KUKA KRL program: MyProgram_089().src

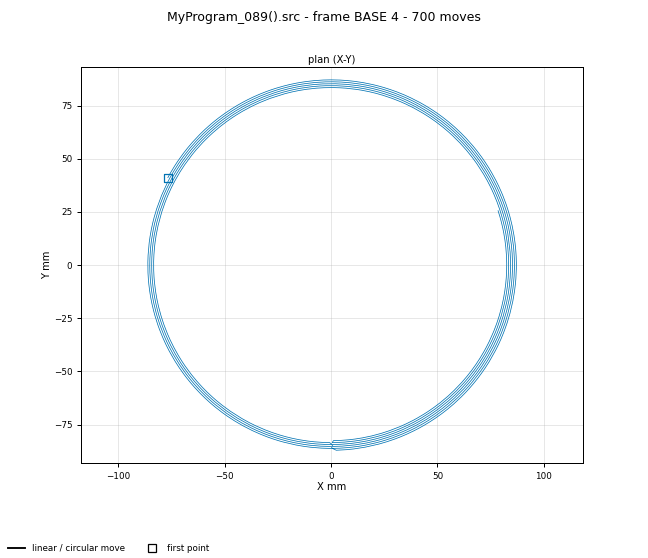
[picture p0: tool path of MyProgram_089().src in frame BASE 4, 700 of 700 moves have a stored position in this frame; points joined in program order, loops and branches not executed]
&ACCESS RVP
&REL 1
&PARAM TEMPLATE = C:\KRC\Roboter\Template\vorgabe
&PARAM EDITMASK = *
DEF MyProgram_089()
; ---- Setting reference (Base) ----
$BASE = BASE_DATA[4]

; --------------------------
; ---- Setting tool (TCP) ----
$TOOL = TOOL_DATA[3]
; --------------------------

$VEL.CP = VEL_APROX_PRINT
Startdeposition()
$VEL.CP = VEL_PRINT
LIN {X -76.7634,Y 41.1633,Z 86,A 146.3137,B 24.9093,C -2.1993,E1 24.8592,E2 298.6214} C_DIS
LIN {X -75.415,Y 43.5831,Z 86,A 144.1649,B 24.9096,C -2.1954,E1 24.8622,E2 300.7907} C_DIS
LIN {X -73.5045,Y 46.7342,Z 86,A 141.7026,B 24.9091,C -2.2011,E1 24.8658,E2 303.2518} C_DIS
LIN {X -72.1353,Y 48.8195,Z 86,A 139.243,B 24.9106,C -2.1828,E1 24.8698,E2 305.7674} C_DIS
LIN {X -69.4773,Y 52.5341,Z 86,A 137.1661,B 24.9078,C -2.2168,E1 24.8731,E2 307.7732} C_DIS
LIN {X -67.5267,Y 55.0186,Z 86,A 134.9351,B 24.9078,C -2.2179,E1 24.877,E2 310.012} C_DIS
LIN {X -65.1327,Y 57.8335,Z 86,A 132.6257,B 24.9069,C -2.2275,E1 24.8812,E2 312.3089} C_DIS
LIN {X -61.7541,Y 61.4278,Z 86,A 128.7956,B 24.9076,C -2.2188,E1 24.8887,E2 316.1763} C_DIS
LIN {X -59.3206,Y 63.7821,Z 86,A 127.0883,B 24.906,C -2.2388,E1 24.8921,E2 317.843} C_DIS
LIN {X -57.1612,Y 65.7228,Z 86,A 125.1507,B 24.9057,C -2.2423,E1 24.8962,E2 319.7798} C_DIS
LIN {X -54.8255,Y 67.6833,Z 86,A 123.2348,B 24.9051,C -2.2493,E1 24.9003,E2 321.6865} C_DIS
LIN {X -52.7347,Y 69.3257,Z 86,A 120.98,B 24.906,C -2.2384,E1 24.9054,E2 323.9752} C_DIS
LIN {X -49.8675,Y 71.4151,Z 86,A 118.3983,B 24.9062,C -2.236,E1 24.9113,E2 326.5717} C_DIS
LIN {X -46.7307,Y 73.5068,Z 86,A 116.0354,B 24.9055,C -2.244,E1 24.9168,E2 328.923} C_DIS
LIN {X -43.9125,Y 75.2237,Z 86,A 114.6023,B 24.9034,C -2.2693,E1 24.9202,E2 330.3002} C_DIS
LIN {X -41.4126,Y 76.6281,Z 86,A 112.4064,B 24.9039,C -2.2635,E1 24.9256,E2 332.5163} C_DIS
LIN {X -39.1074,Y 77.8311,Z 86,A 110.8125,B 24.9034,C -2.2696,E1 24.9295,E2 334.0999} C_DIS
LIN {X -36.432,Y 79.1182,Z 86,A 108.8082,B 24.9032,C -2.2711,E1 24.9346,E2 336.1056} C_DIS
LIN {X -33.5337,Y 80.3893,Z 86,A 106.7104,B 24.903,C -2.2736,E1 24.94,E2 338.2023} C_DIS
LIN {X -30.5403,Y 81.5736,Z 86,A 104.5603,B 24.9029,C -2.2755,E1 24.9456,E2 340.3526} C_DIS
LIN {X -28.173,Y 82.4213,Z 86,A 102.9203,B 24.9027,C -2.2779,E1 24.9499,E2 341.99} C_DIS
LIN {X -25.7542,Y 83.208,Z 86,A 101.1907,B 24.9027,C -2.2782,E1 24.9545,E2 343.722} C_DIS
LIN {X -22.1455,Y 84.2417,Z 86,A 98.7036,B 24.9025,C -2.2802,E1 24.9612,E2 346.2083} C_DIS
LIN {X -19.3941,Y 84.9162,Z 86,A 96.8617,B 24.9023,C -2.2825,E1 24.9662,E2 348.047} C_DIS
LIN {X -16.2854,Y 85.5668,Z 86,A 94.5826,B 24.9026,C -2.2785,E1 24.9725,E2 350.3382} C_DIS
LIN {X -12.7065,Y 86.172,Z 86,A 91.9605,B 24.9031,C -2.2731,E1 24.9797,E2 352.9755} C_DIS
LIN {X -8.1409,Y 86.7214,Z 86,A 89.5155,B 24.9014,C -2.2923,E1 24.9864,E2 355.3763} C_DIS
LIN {X -3.6843,Y 87.0246,Z 86,A 86.4266,B 24.9017,C -2.2888,E1 24.995,E2 358.4744} C_DIS
LIN {X 0.0247,Y 87.104,Z 86,A 83.8791,B 24.902,C -2.286,E1 25.0022,E2 361.0285} C_DIS
LIN {X 4.2369,Y 87.0001,Z 86,A 81.1959,B 24.9017,C -2.289,E1 25.0096,E2 363.7041} C_DIS
LIN {X 7.415,Y 86.7877,Z 86,A 78.9957,B 24.902,C -2.2856,E1 25.0158,E2 365.9111} C_DIS
LIN {X 11.0675,Y 86.3966,Z 86,A 76.481,B 24.9023,C -2.2822,E1 25.0228,E2 368.4322} C_DIS
LIN {X 15.0741,Y 85.789,Z 86,A 73.7549,B 24.9025,C -2.2794,E1 25.0303,E2 371.1621} C_DIS
LIN {X 19.4788,Y 84.8967,Z 86,A 71.0686,B 24.9019,C -2.2864,E1 25.0376,E2 373.8282} C_DIS
LIN {X 22.3755,Y 84.1802,Z 86,A 69.4228,B 24.9012,C -2.2953,E1 25.042,E2 375.4505} C_DIS
LIN {X 24.9228,Y 83.461,Z 86,A 67.479,B 24.9018,C -2.2876,E1 25.0472,E2 377.4091} C_DIS
LIN {X 27.8212,Y 82.5399,Z 86,A 65.4884,B 24.9019,C -2.2864,E1 25.0525,E2 379.399} C_DIS
LIN {X 30.9983,Y 81.4001,Z 86,A 63.1184,B 24.9025,C -2.2795,E1 25.0587,E2 381.7802} C_DIS
LIN {X 34.3976,Y 80.0241,Z 86,A 60.7222,B 24.9027,C -2.2775,E1 25.0649,E2 384.1756} C_DIS
LIN {X 37.4722,Y 78.6306,Z 86,A 58.5492,B 24.9027,C -2.2764,E1 25.0704,E2 386.3456} C_DIS
LIN {X 41.8101,Y 76.4125,Z 86,A 55.3258,B 24.9032,C -2.2716,E1 25.0784,E2 389.5714} C_DIS
LIN {X 45.0669,Y 74.5377,Z 86,A 53.0034,B 24.9031,C -2.2729,E1 25.0839,E2 391.8836} C_DIS
LIN {X 47.6981,Y 72.8823,Z 86,A 50.901,B 24.9035,C -2.2679,E1 25.0889,E2 393.9911} C_DIS
LIN {X 50.5181,Y 70.9562,Z 86,A 48.7009,B 24.9037,C -2.2657,E1 25.0939,E2 396.1888} C_DIS
LIN {X 52.437,Y 69.5502,Z 86,A 46.5187,B 24.9056,C -2.2427,E1 25.0989,E2 398.4176} C_DIS
LIN {X 55.2509,Y 67.3384,Z 86,A 44.6477,B 24.9047,C -2.2541,E1 25.1029,E2 400.2545} C_DIS
LIN {X 58.0486,Y 64.9401,Z 86,A 42.4392,B 24.9045,C -2.2566,E1 25.1075,E2 402.4484} C_DIS
LIN {X 61.0298,Y 62.1472,Z 86,A 39.1117,B 24.9067,C -2.2298,E1 25.1143,E2 405.8255} C_DIS
LIN {X 63.4116,Y 59.7146,Z 86,A 36.9778,B 24.9068,C -2.2284,E1 25.1184,E2 407.9534} C_DIS
LIN {X 66.661,Y 56.0663,Z 86,A 34.1325,B 24.9064,C -2.2333,E1 25.1235,E2 410.7742} C_DIS
LIN {X 68.5605,Y 53.7256,Z 86,A 32.4833,B 24.9059,C -2.2399,E1 25.1264,E2 412.4002} C_DIS
LIN {X 70.7515,Y 50.805,Z 86,A 30.1365,B 24.9062,C -2.2359,E1 25.1303,E2 414.7453} C_DIS
LIN {X 72.2333,Y 48.6749,Z 86,A 28.14,B 24.9074,C -2.2217,E1 25.1335,E2 416.7653} C_DIS
LIN {X 74.1305,Y 45.7351,Z 86,A 25.9158,B 24.9077,C -2.2184,E1 25.1368,E2 418.9861} C_DIS
LIN {X 75.4436,Y 43.5333,Z 86,A 24.1981,B 24.9081,C -2.2129,E1 25.1392,E2 420.7081} C_DIS
LIN {X 77.4348,Y 39.8846,Z 86,A 21.5317,B 24.9086,C -2.2077,E1 25.1427,E2 423.3726} C_DIS
LIN {X 78.666,Y 37.3985,Z 86,A 19.6238,B 24.9092,C -2.1998,E1 25.145,E2 425.289} C_DIS
LIN {X 80.0248,Y 34.3961,Z 86,A 17.5675,B 24.9094,C -2.1974,E1 25.1474,E2 427.3396} C_DIS
LIN {X 80.8251,Y 32.4701,Z 86,A 15.9985,B 24.9103,C -2.1867,E1 25.149,E2 428.9252} C_DIS
LIN {X 82.1991,Y 28.8126,Z 86,A 13.5608,B 24.9106,C -2.1838,E1 25.1513,E2 431.3563} C_DIS
LIN {X 83.2983,Y 25.4632,Z 86,A 11.4352,B 24.9106,C -2.1835,E1 25.1531,E2 433.4705} C_DIS
LIN {X 84.1421,Y 22.5169,Z 86,A 9.258,B 24.9115,C -2.1718,E1 25.1548,E2 435.6627} C_DIS
LIN {X 85.1237,Y 18.4612,Z 86,A 6.1814,B 24.9131,C -2.152,E1 25.1567,E2 438.7683} C_DIS
LIN {X 85.9827,Y 13.9294,Z 86,A 3.4164,B 24.9131,C -2.1518,E1 25.158,E2 441.5175} C_DIS
LIN {X 86.4939,Y 10.2803,Z 86,A 1.1857,B 24.9132,C -2.1509,E1 25.1588,E2 443.7373} C_DIS
LIN {X 86.8107,Y 7.1264,Z 86,A -0.8981,B 24.9138,C -2.1443,E1 25.1594,E2 445.8242} C_DIS
LIN {X 87.0169,Y 3.8645,Z 86,A -2.9324,B 24.914,C -2.1415,E1 25.1597,E2 447.853} C_DIS
LIN {X 87.0973,Y 1.0892,Z 86,A -5.0184,B 24.9152,C -2.1266,E1 25.1597,E2 449.9617} C_DIS
LIN {X 87.0851,Y -1.7482,Z 86,A -6.7904,B 24.9154,C -2.124,E1 25.1597,E2 451.7295} C_DIS
LIN {X 86.8701,Y -6.3796,Z 86,A -9.6702,B 24.9157,C -2.12,E1 25.1593,E2 454.6014} C_DIS
LIN {X 86.6351,Y -9.012,Z 86,A -11.4896,B 24.9164,C -2.1117,E1 25.1588,E2 456.4298} C_DIS
LIN {X 86.2143,Y -12.4087,Z 86,A -14.6166,B 24.9193,C -2.0744,E1 25.1575,E2 459.6264} C_DIS
LIN {X 85.4298,Y -16.9968,Z 86,A -16.5812,B 24.9171,C -2.1024,E1 25.1566,E2 461.5134} C_DIS
LIN {X 84.1155,Y -22.6153,Z 86,A -20.4328,B 24.9182,C -2.0884,E1 25.154,E2 465.3757} C_DIS
LIN {X 82.7404,Y -27.2225,Z 86,A -24.1318,B 24.9204,C -2.06,E1 25.1509,E2 469.1206} C_DIS
LIN {X 81.1349,Y -31.6862,Z 86,A -26.741,B 24.9198,C -2.0681,E1 25.1484,E2 471.6962} C_DIS
LIN {X 79.8438,Y -34.8112,Z 86,A -29.0086,B 24.9204,C -2.0598,E1 25.1459,E2 473.9709} C_DIS
LIN {X 78.7096,Y -37.3077,Z 86,A -30.8316,B 24.9209,C -2.0538,E1 25.1437,E2 475.7984} C_DIS
LIN {X 77.2971,Y -40.1528,Z 86,A -33.0905,B 24.9218,C -2.0418,E1 25.1409,E2 478.0737} C_DIS
LIN {X 74.3275,Y -45.4128,Z 86,A -36.9909,B 24.9225,C -2.0329,E1 25.1354,E2 481.975} C_DIS
LIN {X 72.2956,Y -48.5828,Z 86,A -39.2144,B 24.9224,C -2.0346,E1 25.132,E2 484.1832} C_DIS
LIN {X 70.6239,Y -50.9837,Z 86,A -41.1745,B 24.9229,C -2.0281,E1 25.1288,E2 486.1491} C_DIS
LIN {X 68.7131,Y -53.531,Z 86,A -43.1701,B 24.923,C -2.0259,E1 25.1254,E2 488.1404} C_DIS
LIN {X 66.9112,Y -55.7652,Z 86,A -45.1338,B 24.9236,C -2.0184,E1 25.1219,E2 490.1128} C_DIS
LIN {X 64.7202,Y -58.2943,Z 86,A -47.3545,B 24.9241,C -2.0121,E1 25.1178,E2 492.3384} C_DIS
LIN {X 62.938,Y -60.2143,Z 86,A -49.1674,B 24.9246,C -2.0048,E1 25.1143,E2 494.1607} C_DIS
LIN {X 61.1438,Y -62.0347,Z 86,A -51.6966,B 24.9271,C -1.9722,E1 25.1092,E2 496.7563} C_DIS
LIN {X 57.5449,Y -65.3877,Z 86,A -53.9194,B 24.9251,C -1.9987,E1 25.1047,E2 498.9075} C_DIS
LIN {X 55.0102,Y -67.5335,Z 86,A -55.8925,B 24.9249,C -2.001,E1 25.1005,E2 500.8676} C_DIS
LIN {X 53.3581,Y -68.8464,Z 86,A -57.4566,B 24.9256,C -1.9921,E1 25.097,E2 502.447} C_DIS
LIN {X 51.5911,Y -70.1801,Z 86,A -58.8812,B 24.9257,C -1.9901,E1 25.0938,E2 503.8712} C_DIS
LIN {X 48.9288,Y -72.0614,Z 86,A -60.9649,B 24.9259,C -1.9879,E1 25.089,E2 505.9531} C_DIS
LIN {X 46.5742,Y -73.6067,Z 86,A -62.9319,B 24.9265,C -1.9804,E1 25.0844,E2 507.9313} C_DIS
LIN {X 43.8648,Y -75.2527,Z 86,A -64.9876,B 24.9267,C -1.9776,E1 25.0795,E2 509.9874} C_DIS
LIN {X 41.2059,Y -76.7396,Z 86,A -66.9966,B 24.9269,C -1.974,E1 25.0745,E2 511.9992} C_DIS
LIN {X 38.8987,Y -77.9346,Z 86,A -69.3028,B 24.9286,C -1.9515,E1 25.0687,E2 514.3523} C_DIS
LIN {X 35.5869,Y -79.5014,Z 86,A -71.5732,B 24.9286,C -1.9524,E1 25.0629,E2 516.615} C_DIS
LIN {X 32.616,Y -80.7656,Z 86,A -73.1461,B 24.9274,C -1.9674,E1 25.0589,E2 518.1486} C_DIS
LIN {X 29.7282,Y -81.8725,Z 86,A -75.2929,B 24.9279,C -1.961,E1 25.0533,E2 520.306} C_DIS
LIN {X 26.2462,Y -83.0555,Z 86,A -77.5924,B 24.9279,C -1.962,E1 25.0472,E2 522.5989} C_DIS
LIN {X 22.4058,Y -84.1721,Z 86,A -80.4955,B 24.9287,C -1.9503,E1 25.0393,E2 525.5249} C_DIS
LIN {X 16.0344,Y -85.6151,Z 86,A -84.4685,B 24.9282,C -1.9569,E1 25.0286,E2 529.4771} C_DIS
LIN {X 10.7051,Y -86.4436,Z 86,A -88.1837,B 24.9288,C -1.949,E1 25.0182,E2 533.2075} C_DIS
LIN {X 7.4273,Y -86.7867,Z 86,A -90.3524,B 24.9288,C -1.9479,E1 25.0122,E2 535.3777} C_DIS
LIN {X 2.4408,Y -87.0687,Z 86,A -93.6388,B 24.929,C -1.9466,E1 25.003,E2 538.6661} C_DIS
LIN {X 2.4408,Y -87.0687,Z 86,A -93.6388,B 24.929,C -1.9466,E1 25.003,E2 538.6661} C_DIS
Enddeposition()
LIN {X 0.5553,Y -86.1888,Z 86,A -93.3756,B 24.9242,C -2.0102,E1 25.0042,E2 538.2522} C_DIS
Startdeposition()
$VEL.CP = VEL_PRINT
LIN {X 3.8721,Y -86.1086,Z 86,A -91.75,B 24.9256,C -1.9922,E1 25.0086,E2 536.6696} C_DIS
LIN {X 8.5981,Y -85.7663,Z 86,A -88.5017,B 24.9252,C -1.9969,E1 25.0177,E2 533.4119} C_DIS
LIN {X 13.0459,Y -85.2026,Z 86,A -85.1686,B 24.9242,C -2.0103,E1 25.027,E2 530.0497} C_DIS
LIN {X 16.2421,Y -84.6514,Z 86,A -82.1799,B 24.922,C -2.0396,E1 25.0354,E2 526.9952} C_DIS
LIN {X 21.4948,Y -83.4723,Z 86,A -80.2349,B 24.9258,C -1.9893,E1 25.0403,E2 525.1723} C_DIS
LIN {X 24.1077,Y -82.7557,Z 86,A -78.0283,B 24.9247,C -2.0045,E1 25.0463,E2 522.9333} C_DIS
LIN {X 26.2649,Y -82.0969,Z 86,A -76.4934,B 24.9244,C -2.0074,E1 25.0504,E2 521.3943} C_DIS
LIN {X 29.1197,Y -81.1289,Z 86,A -74.3708,B 24.924,C -2.0139,E1 25.056,E2 519.2606} C_DIS
LIN {X 33.6141,Y -79.3711,Z 86,A -71.1979,B 24.9237,C -2.0173,E1 25.0642,E2 516.087} C_DIS
LIN {X 37.2598,Y -77.7263,Z 86,A -68.3723,B 24.923,C -2.027,E1 25.0714,E2 513.2456} C_DIS
LIN {X 39.8478,Y -76.4326,Z 86,A -65.8675,B 24.9212,C -2.0498,E1 25.0778,E2 510.6938} C_DIS
LIN {X 43.6555,Y -74.323,Z 86,A -63.7162,B 24.9227,C -2.0299,E1 25.0828,E2 508.5961} C_DIS
LIN {X 46.5967,Y -72.5149,Z 86,A -61.6607,B 24.923,C -2.0262,E1 25.0876,E2 506.556} C_DIS
LIN {X 49.1239,Y -70.8273,Z 86,A -59.6458,B 24.9227,C -2.03,E1 25.0923,E2 504.5388} C_DIS
LIN {X 52.7293,Y -68.1858,Z 86,A -56.395,B 24.9215,C -2.0457,E1 25.0996,E2 501.2625} C_DIS
LIN {X 55.5568,Y -65.9038,Z 86,A -54.1006,B 24.9215,C -2.047,E1 25.1045,E2 498.9741} C_DIS
LIN {X 59.5946,Y -62.2747,Z 86,A -50.5714,B 24.921,C -2.0526,E1 25.1118,E2 495.4456} C_DIS
LIN {X 62.0674,Y -59.8105,Z 86,A -48.2048,B 24.9204,C -2.0599,E1 25.1164,E2 493.0721} C_DIS
LIN {X 64.5863,Y -57.0836,Z 86,A -45.8968,B 24.9204,C -2.0606,E1 25.1207,E2 490.7727} C_DIS
LIN {X 66.5451,Y -54.7865,Z 86,A -43.5845,B 24.9192,C -2.0764,E1 25.1249,E2 488.4338} C_DIS
LIN {X 70.0716,Y -50.1962,Z 86,A -40.0232,B 24.9192,C -2.0768,E1 25.1309,E2 484.8884} C_DIS
LIN {X 71.8513,Y -47.614,Z 86,A -37.3481,B 24.917,C -2.1031,E1 25.1351,E2 482.1645} C_DIS
LIN {X 73.7236,Y -44.6599,Z 86,A -35.9077,B 24.9189,C -2.079,E1 25.1371,E2 480.7883} C_DIS
LIN {X 76.3659,Y -39.9744,Z 86,A -32.2618,B 24.9179,C -2.0918,E1 25.1421,E2 477.1312} C_DIS
LIN {X 77.7306,Y -37.2508,Z 86,A -30.1507,B 24.9172,C -2.1008,E1 25.1447,E2 475.0102} C_DIS
LIN {X 79.2268,Y -33.9566,Z 86,A -27.6767,B 24.9165,C -2.1104,E1 25.1475,E2 472.527} C_DIS
LIN {X 80.2416,Y -31.4792,Z 86,A -25.4793,B 24.9149,C -2.1304,E1 25.1498,E2 470.2944} C_DIS
LIN {X 81.841,Y -27.055,Z 86,A -22.658,B 24.9149,C -2.1294,E1 25.1523,E2 467.4915} C_DIS
LIN {X 82.9666,Y -23.3714,Z 86,A -20.3616,B 24.9151,C -2.1282,E1 25.1541,E2 465.211} C_DIS
LIN {X 84.489,Y -17.0685,Z 86,A -16.1871,B 24.9143,C -2.137,E1 25.1568,E2 461.0398} C_DIS
LIN {X 85.4391,Y -11.3985,Z 86,A -12.4656,B 24.9137,C -2.1457,E1 25.1585,E2 457.3197} C_DIS
LIN {X 85.8101,Y -8.1449,Z 86,A -9.8442,B 24.9118,C -2.1681,E1 25.1593,E2 454.6609} C_DIS
LIN {X 86.0443,Y -5.1157,Z 86,A -7.3413,B 24.9099,C -2.1916,E1 25.1597,E2 452.1175} C_DIS
LIN {X 86.1848,Y -1.3715,Z 86,A -5.5151,B 24.9112,C -2.1762,E1 25.1597,E2 450.3384} C_DIS
LIN {X 86.1382,Y 3.1833,Z 86,A -2.2209,B 24.9096,C -2.1952,E1 25.1596,E2 447.0191} C_DIS
LIN {X 85.9696,Y 6.2509,Z 86,A -0.4717,B 24.9099,C -2.1914,E1 25.1592,E2 445.2891} C_DIS
LIN {X 85.6888,Y 9.3393,Z 86,A 1.541,B 24.9095,C -2.1962,E1 25.1587,E2 443.277} C_DIS
LIN {X 84.8873,Y 14.9631,Z 86,A 4.9917,B 24.9095,C -2.1967,E1 25.1573,E2 439.8454} C_DIS
LIN {X 83.9417,Y 19.5828,Z 86,A 7.9872,B 24.9091,C -2.2016,E1 25.1556,E2 436.8559} C_DIS
LIN {X 83.4156,Y 21.7157,Z 86,A 9.9382,B 24.9073,C -2.223,E1 25.1542,E2 434.8657} C_DIS
LIN {X 82.4756,Y 25.0536,Z 86,A 12.208,B 24.9068,C -2.2287,E1 25.1524,E2 432.5955} C_DIS
LIN {X 81.485,Y 28.1081,Z 86,A 14.3003,B 24.9064,C -2.2335,E1 25.1506,E2 430.5035} C_DIS
LIN {X 80.715,Y 30.2464,Z 86,A 16.6699,B 24.9035,C -2.2678,E1 25.1482,E2 428.0662} C_DIS
LIN {X 79.0291,Y 34.4103,Z 86,A 18.6301,B 24.9058,C -2.2408,E1 25.1461,E2 426.1805} C_DIS
LIN {X 77.8734,Y 36.9535,Z 86,A 21.6178,B 24.902,C -2.285,E1 25.1424,E2 423.1043} C_DIS
LIN {X 75.6326,Y 41.3454,Z 86,A 23.855,B 24.9044,C -2.258,E1 25.1395,E2 420.9428} C_DIS
LIN {X 74.0596,Y 44.1012,Z 86,A 26.2172,B 24.9031,C -2.2722,E1 25.1362,E2 418.559} C_DIS
LIN {X 72.0182,Y 47.3609,Z 86,A 28.3952,B 24.9037,C -2.2659,E1 25.1329,E2 416.4069} C_DIS
LIN {X 70.4033,Y 49.7312,Z 86,A 30.7155,B 24.9021,C -2.2848,E1 25.1291,E2 414.0535} C_DIS
LIN {X 67.5766,Y 53.5076,Z 86,A 33.5411,B 24.9023,C -2.2818,E1 25.1244,E2 411.2482} C_DIS
LIN {X 65.6319,Y 55.8759,Z 86,A 35.6341,B 24.9018,C -2.2884,E1 25.1206,E2 409.1492} C_DIS
LIN {X 61.1648,Y 60.7336,Z 86,A 39.729,B 24.9018,C -2.2882,E1 25.1128,E2 405.0727} C_DIS
LIN {X 59.7975,Y 62.0799,Z 86,A 41.3725,B 24.9005,C -2.3031,E1 25.1095,E2 403.4007} C_DIS
LIN {X 56.9904,Y 64.6676,Z 86,A 43.7106,B 24.9006,C -2.3015,E1 25.1046,E2 401.0759} C_DIS
LIN {X 54.6012,Y 66.6975,Z 86,A 46.2078,B 24.8991,C -2.3192,E1 25.0992,E2 398.5463} C_DIS
LIN {X 50.4399,Y 69.8976,Z 86,A 49.1243,B 24.9002,C -2.3063,E1 25.0928,E2 395.6709} C_DIS
LIN {X 47.8883,Y 71.6705,Z 86,A 51.2386,B 24.8998,C -2.3112,E1 25.0879,E2 393.552} C_DIS
LIN {X 45.1615,Y 73.4187,Z 86,A 53.8543,B 24.8982,C -2.3298,E1 25.0816,E2 390.9008} C_DIS
LIN {X 41.1371,Y 75.7456,Z 86,A 57.0566,B 24.8975,C -2.3377,E1 25.0738,E2 387.689} C_DIS
LIN {X 38.1933,Y 77.2719,Z 86,A 59.235,B 24.8973,C -2.3396,E1 25.0683,E2 385.512} C_DIS
LIN {X 35.2475,Y 78.6594,Z 86,A 60.7706,B 24.8989,C -2.3216,E1 25.0645,E2 384.0229} C_DIS
LIN {X 30.2889,Y 80.6989,Z 86,A 64.5187,B 24.898,C -2.3311,E1 25.0548,E2 380.2607} C_DIS
LIN {X 26.7118,Y 81.9523,Z 86,A 66.9481,B 24.8981,C -2.3303,E1 25.0484,E2 377.838} C_DIS
LIN {X 23.5489,Y 82.9163,Z 86,A 69.1096,B 24.8981,C -2.3307,E1 25.0426,E2 375.6792} C_DIS
LIN {X 20.0579,Y 83.8301,Z 86,A 71.5045,B 24.898,C -2.332,E1 25.0361,E2 373.2849} C_DIS
LIN {X 16.8841,Y 84.5269,Z 86,A 74.238,B 24.8963,C -2.3512,E1 25.0285,E2 370.5092} C_DIS
LIN {X 13.6155,Y 85.1145,Z 86,A 76.0994,B 24.8972,C -2.3409,E1 25.0234,E2 368.674} C_DIS
LIN {X 9.149,Y 85.7087,Z 86,A 78.519,B 24.8987,C -2.3235,E1 25.0169,E2 366.2978} C_DIS
LIN {X 4.6296,Y 86.0711,Z 86,A 81.8771,B 24.8978,C -2.3343,E1 25.0074,E2 362.9155} C_DIS
LIN {X 0.939,Y 86.1897,Z 86,A 84.7013,B 24.8968,C -2.3455,E1 24.9995,E2 360.0652} C_DIS
LIN {X -2.6768,Y 86.1539,Z 86,A 86.8743,B 24.8975,C -2.3377,E1 24.9935,E2 357.9106} C_DIS
LIN {X -7.7582,Y 85.8458,Z 86,A 89.7735,B 24.8989,C -2.3214,E1 24.9855,E2 355.0489} C_DIS
LIN {X -12.4441,Y 85.2931,Z 86,A 93.1212,B 24.8985,C -2.3259,E1 24.9762,E2 351.6881} C_DIS
LIN {X -14.9601,Y 84.8878,Z 86,A 94.9954,B 24.8981,C -2.3302,E1 24.971,E2 349.8021} C_DIS
LIN {X -18.1469,Y 84.2639,Z 86,A 97.1348,B 24.8983,C -2.3278,E1 24.9651,E2 347.6658} C_DIS
LIN {X -21.1295,Y 83.5662,Z 86,A 99.1946,B 24.8984,C -2.3266,E1 24.9596,E2 345.6061} C_DIS
LIN {X -24.0255,Y 82.781,Z 86,A 101.3524,B 24.8982,C -2.3294,E1 24.9537,E2 343.4382} C_DIS
LIN {X -26.6719,Y 81.9652,Z 86,A 103.5921,B 24.8973,C -2.3393,E1 24.9477,E2 341.1709} C_DIS
LIN {X -29.8506,Y 80.8623,Z 86,A 105.0252,B 24.8997,C -2.3124,E1 24.9441,E2 339.7989} C_DIS
LIN {X -33.387,Y 79.4668,Z 86,A 107.7798,B 24.8994,C -2.3157,E1 24.9369,E2 337.0305} C_DIS
LIN {X -36.226,Y 78.2136,Z 86,A 110.2294,B 24.8987,C -2.324,E1 24.9306,E2 334.5549} C_DIS
LIN {X -39.9,Y 76.4051,Z 86,A 112.6449,B 24.8998,C -2.3106,E1 24.9247,E2 332.1649} C_DIS
LIN {X -42.7024,Y 74.8748,Z 86,A 114.9169,B 24.8998,C -2.3113,E1 24.9191,E2 329.8846} C_DIS
LIN {X -46.4038,Y 72.6387,Z 86,A 117.9459,B 24.8998,C -2.3105,E1 24.9119,E2 326.848} C_DIS
LIN {X -50.3519,Y 69.9605,Z 86,A 121.2138,B 24.9001,C -2.307,E1 24.9045,E2 323.5773} C_DIS
LIN {X -53.9354,Y 67.2371,Z 86,A 124.0774,B 24.901,C -2.2969,E1 24.8982,E2 320.7271} C_DIS
LIN {X -57.9428,Y 63.8161,Z 86,A 127.9034,B 24.9009,C -2.2984,E1 24.8902,E2 316.8825} C_DIS
LIN {X -60.3048,Y 61.5865,Z 86,A 129.7077,B 24.9022,C -2.283,E1 24.8866,E2 315.1073} C_DIS
LIN {X -63.3063,Y 58.4954,Z 86,A 132.768,B 24.9023,C -2.2816,E1 24.8807,E2 312.0369} C_DIS
LIN {X -66.4209,Y 54.936,Z 86,A 135.8403,B 24.9032,C -2.2715,E1 24.8752,E2 308.9748} C_DIS
LIN {X -69.3278,Y 51.2196,Z 86,A 139.1812,B 24.9034,C -2.269,E1 24.8696,E2 305.6239} C_DIS
LIN {X -71.7307,Y 47.7969,Z 86,A 141.7923,B 24.9045,C -2.2565,E1 24.8655,E2 303.0296} C_DIS
LIN {X -74.0479,Y 44.1209,Z 86,A 144.4199,B 24.9058,C -2.2409,E1 24.8617,E2 300.4256} C_DIS
LIN {X -75.5519,Y 41.4942,Z 86,A 146.4376,B 24.9063,C -2.2353,E1 24.8589,E2 298.4108} C_DIS
LIN {X -77.1803,Y 38.3781,Z 86,A 149.1153,B 24.906,C -2.2381,E1 24.8555,E2 295.7122} C_DIS
LIN {X -79.6902,Y 32.8523,Z 86,A 152.9138,B 24.9076,C -2.2193,E1 24.8513,E2 291.9377} C_DIS
LIN {X -82.0216,Y 26.4975,Z 86,A 157.3186,B 24.909,C -2.2027,E1 24.8472,E2 287.5473} C_DIS
LIN {X -83.2516,Y 22.3349,Z 86,A 160.1807,B 24.9098,C -2.1931,E1 24.845,E2 284.6918} C_DIS
LIN {X -83.8659,Y 19.9107,Z 86,A 161.8913,B 24.9101,C -2.1892,E1 24.8438,E2 282.9804} C_DIS
LIN {X -84.5406,Y 16.8172,Z 86,A 164.0758,B 24.9105,C -2.1847,E1 24.8426,E2 280.7937} C_DIS
LIN {X -85.1512,Y 13.3779,Z 86,A 166.3693,B 24.9111,C -2.1766,E1 24.8415,E2 278.506} C_DIS
LIN {X -85.5596,Y 10.4597,Z 86,A 168.8152,B 24.9105,C -2.184,E1 24.8407,E2 276.0278} C_DIS
LIN {X -86.0761,Y 4.5397,Z 86,A 172.468,B 24.9122,C -2.163,E1 24.8399,E2 272.4032} C_DIS
LIN {X -86.1868,Y 1.2662,Z 86,A 174.9812,B 24.912,C -2.1655,E1 24.8398,E2 269.8688} C_DIS
LIN {X -86.1179,Y -3.6564,Z 86,A 177.7256,B 24.9141,C -2.1402,E1 24.84,E2 267.1683} C_DIS
LIN {X -85.9343,Y -6.7062,Z 86,A 179.531,B 24.9151,C -2.1275,E1 24.8403,E2 265.3824} C_DIS
LIN {X -85.7225,Y -9.0176,Z 86,A -178.321,B 24.9141,C -2.1396,E1 24.8409,E2 263.1927} C_DIS
LIN {X -85.3543,Y -12.0133,Z 86,A -176.5494,B 24.9152,C -2.1267,E1 24.8416,E2 261.4412} C_DIS
LIN {X -84.8694,Y -15.0628,Z 86,A -174.5012,B 24.9157,C -2.1202,E1 24.8425,E2 259.3964} C_DIS
LIN {X -84.2966,Y -17.997,Z 86,A -172.3818,B 24.9159,C -2.1178,E1 24.8437,E2 257.2703} C_DIS
LIN {X -83.5833,Y -21.0633,Z 86,A -170.3524,B 24.9165,C -2.1096,E1 24.845,E2 255.2486} C_DIS
LIN {X -82.8564,Y -23.7602,Z 86,A -168.5401,B 24.9171,C -2.1027,E1 24.8464,E2 253.4421} C_DIS
LIN {X -81.5811,Y -27.8257,Z 86,A -165.8313,B 24.918,C -2.0908,E1 24.8487,E2 250.7461} C_DIS
LIN {X -80.6988,Y -30.2891,Z 86,A -163.4949,B 24.9171,C -2.1027,E1 24.851,E2 248.3682} C_DIS
LIN {X -79.0848,Y -34.2824,Z 86,A -160.9313,B 24.9184,C -2.086,E1 24.8537,E2 245.8303} C_DIS
LIN {X -77.66,Y -37.3977,Z 86,A -158.709,B 24.919,C -2.078,E1 24.8564,E2 243.6149} C_DIS
LIN {X -76.0791,Y -40.5191,Z 86,A -156.2198,B 24.9192,C -2.0764,E1 24.8596,E2 241.1164} C_DIS
LIN {X -73.3035,Y -45.3475,Z 86,A -152.5489,B 24.92,C -2.0657,E1 24.8648,E2 237.452} C_DIS
LIN {X -71.4037,Y -48.2823,Z 86,A -149.5854,B 24.919,C -2.0784,E1 24.8695,E2 234.4433} C_DIS
LIN {X -69.1658,Y -51.4386,Z 86,A -147.9305,B 24.9215,C -2.0454,E1 24.8721,E2 232.8591} C_DIS
LIN {X -67.8726,Y -53.1331,Z 86,A -146.283,B 24.9213,C -2.0487,E1 24.8749,E2 231.1959} C_DIS
LIN {X -66.0712,Y -55.3569,Z 86,A -144.4081,B 24.9217,C -2.0435,E1 24.8782,E2 229.3247} C_DIS
LIN {X -64.149,Y -57.5724,Z 86,A -142.1609,B 24.9214,C -2.0478,E1 24.8824,E2 227.0571} C_DIS
LIN {X -61.8419,Y -60.0445,Z 86,A -140.0048,B 24.9219,C -2.0403,E1 24.8866,E2 224.9097} C_DIS
LIN {X -59.1443,Y -62.7026,Z 86,A -137.6562,B 24.9227,C -2.0302,E1 24.8913,E2 222.5755} C_DIS
LIN {X -56.9275,Y -64.7226,Z 86,A -135.6333,B 24.9229,C -2.0271,E1 24.8955,E2 220.5518} C_DIS
LIN {X -54.6919,Y -66.6235,Z 86,A -133.162,B 24.922,C -2.0389,E1 24.9009,E2 218.0429} C_DIS
LIN {X -51.3251,Y -69.2506,Z 86,A -130.7507,B 24.9234,C -2.0212,E1 24.9062,E2 215.6652} C_DIS
LIN {X -48.7319,Y -71.0992,Z 86,A -128.2162,B 24.9227,C -2.0303,E1 24.9121,E2 213.1004} C_DIS
LIN {X -45.396,Y -73.2732,Z 86,A -126.0301,B 24.9241,C -2.0124,E1 24.9171,E2 210.9499} C_DIS
LIN {X -41.5678,Y -75.5116,Z 86,A -122.8318,B 24.9238,C -2.0159,E1 24.925,E2 207.734} C_DIS
LIN {X -37.0249,Y -77.8392,Z 86,A -118.8609,B 24.9228,C -2.0295,E1 24.935,E2 203.7203} C_DIS
LIN {X -33.2317,Y -79.5323,Z 86,A -117.0231,B 24.9251,C -1.9982,E1 24.9396,E2 201.9526} C_DIS
LIN {X -30.004,Y -80.8063,Z 86,A -114.7164,B 24.9253,C -1.9961,E1 24.9456,E2 199.6462} C_DIS
LIN {X -27.1972,Y -81.793,Z 86,A -112.6645,B 24.9253,C -1.9967,E1 24.951,E2 197.5887} C_DIS
LIN {X -24.5686,Y -82.6199,Z 86,A -111.0332,B 24.9258,C -1.9892,E1 24.9553,E2 195.9724} C_DIS
LIN {X -22.4455,Y -83.2218,Z 86,A -109.3372,B 24.9253,C -1.9954,E1 24.9599,E2 194.2592} C_DIS
LIN {X -16.4006,Y -84.6209,Z 86,A -104.5942,B 24.924,C -2.0129,E1 24.973,E2 189.4687} C_DIS
LIN {X -13.011,Y -85.208,Z 86,A -102.9095,B 24.9255,C -1.9933,E1 24.9775,E2 187.8292} C_DIS
LIN {X -9.6911,Y -85.6496,Z 86,A -100.2271,B 24.9244,C -2.0073,E1 24.9851,E2 185.1115} C_DIS
LIN {X -4.4354,Y -86.0819,Z 86,A -97.1375,B 24.9254,C -1.9942,E1 24.9936,E2 182.0521} C_DIS
LIN {X -1.4013,Y -86.1843,Z 86,A -95.1006,B 24.9254,C -1.9951,E1 24.9993,E2 180.0127} C_DIS
LIN {X 0.5553,Y -86.1888,Z 86,A -93.3733,B 24.9243,C -2.0092,E1 25.0042,E2 178.2522} C_DIS
Enddeposition()
LIN {X 0.5553,Y -86.1888,Z 86,A -93.3733,B 24.9243,C -2.0092,E1 25.0042,E2 178.2522} C_DIS
Startdeposition()
$VEL.CP = VEL_PRINT
LIN {X 0.0638,Y -85.2896,Z 86,A -95.0303,B 24.9263,C -1.9827,E1 24.9994,E2 179.9719} C_DIS
LIN {X -4.8185,Y -85.1522,Z 86,A -98.2795,B 24.9263,C -1.9833,E1 24.9903,E2 183.2202} C_DIS
LIN {X -9.8423,Y -84.7186,Z 86,A -101.7537,B 24.9264,C -1.9808,E1 24.9807,E2 186.702} C_DIS
LIN {X -13.052,Y -84.2838,Z 86,A -104.4129,B 24.9275,C -1.9666,E1 24.9732,E2 189.3971} C_DIS
LIN {X -17.5571,Y -83.4627,Z 86,A -107.3505,B 24.9271,C -1.972,E1 24.9652,E2 192.3252} C_DIS
LIN {X -21.0062,Y -82.6614,Z 86,A -109.4522,B 24.9264,C -1.9816,E1 24.9595,E2 194.407} C_DIS
LIN {X -24.1919,Y -81.7855,Z 86,A -111.7583,B 24.9264,C -1.9805,E1 24.9533,E2 196.7195} C_DIS
LIN {X -27.8379,Y -80.6185,Z 86,A -114.0739,B 24.9257,C -1.9902,E1 24.9472,E2 199.0165} C_DIS
LIN {X -31.2159,Y -79.3705,Z 86,A -116.6127,B 24.9258,C -1.9888,E1 24.9406,E2 201.5637} C_DIS
LIN {X -35.0892,Y -77.7358,Z 86,A -119.331,B 24.9254,C -1.9949,E1 24.9336,E2 204.2738} C_DIS
LIN {X -37.3292,Y -76.6866,Z 86,A -121.5443,B 24.9264,C -1.9806,E1 24.9279,E2 206.5268} C_DIS
LIN {X -42.0382,Y -74.2092,Z 86,A -124.8702,B 24.9256,C -1.9926,E1 24.9198,E2 209.8336} C_DIS
LIN {X -45.1121,Y -72.3811,Z 86,A -128.1839,B 24.9272,C -1.97,E1 24.9118,E2 213.2116} C_DIS
LIN {X -49.0863,Y -69.7488,Z 86,A -130.1888,B 24.9243,C -2.0095,E1 24.9074,E2 215.129} C_DIS
LIN {X -54.5258,Y -65.5824,Z 86,A -134.5846,B 24.9232,C -2.0237,E1 24.8977,E2 219.5072} C_DIS
LIN {X -56.2412,Y -64.1176,Z 86,A -136.5962,B 24.9241,C -2.0123,E1 24.8934,E2 221.5537} C_DIS
LIN {X -58.8003,Y -61.781,Z 86,A -139.048,B 24.924,C -2.0135,E1 24.8884,E2 224.0127} C_DIS
LIN {X -61.7393,Y -58.8438,Z 86,A -142.4329,B 24.9248,C -2.0027,E1 24.8817,E2 227.4378} C_DIS
LIN {X -64.3364,Y -55.9907,Z 86,A -144.1581,B 24.9225,C -2.0329,E1 24.8787,E2 229.0989} C_DIS
LIN {X -66.1077,Y -53.8883,Z 86,A -146.1549,B 24.9225,C -2.0329,E1 24.8751,E2 231.1048} C_DIS
LIN {X -68.0446,Y -51.4208,Z 86,A -149.5164,B 24.9248,C -2.0033,E1 24.8693,E2 234.5532} C_DIS
LIN {X -71.2147,Y -46.9316,Z 86,A -151.4819,B 24.9204,C -2.0604,E1 24.8664,E2 236.3921} C_DIS
LIN {X -74.182,Y -42.0876,Z 86,A -156.0004,B 24.9211,C -2.0508,E1 24.8598,E2 240.9568} C_DIS
LIN {X -76.1143,Y -38.4819,Z 86,A -158.4984,B 24.92,C -2.0652,E1 24.8566,E2 243.4338} C_DIS
LIN {X -77.2573,Y -36.131,Z 86,A -160.2995,B 24.9197,C -2.0689,E1 24.8544,E2 245.2359} C_DIS
LIN {X -78.4356,Y -33.4982,Z 86,A -162.3186,B 24.9195,C -2.0721,E1 24.8521,E2 247.2584} C_DIS
LIN {X -80.3764,Y -28.5278,Z 86,A -166.7962,B 24.9206,C -2.0583,E1 24.8477,E2 251.7943} C_DIS
LIN {X -81.7222,Y -24.4051,Z 86,A -168.6787,B 24.9177,C -2.095,E1 24.8463,E2 253.6001} C_DIS
LIN {X -82.4208,Y -21.9324,Z 86,A -170.6054,B 24.9177,C -2.0947,E1 24.8448,E2 255.5386} C_DIS
LIN {X -83.3934,Y -17.8815,Z 86,A -173.5768,B 24.9174,C -2.0985,E1 24.843,E2 258.5182} C_DIS
LIN {X -84.0351,Y -14.5764,Z 86,A -175.6205,B 24.9164,C -2.1115,E1 24.8419,E2 260.5432} C_DIS
LIN {X -84.5081,Y -11.5208,Z 86,A -177.896,B 24.9164,C -2.1126,E1 24.841,E2 262.8296} C_DIS
LIN {X -84.9422,Y -7.6781,Z 86,A 179.6177,B 24.9154,C -2.1238,E1 24.8403,E2 265.304} C_DIS
LIN {X -85.2165,Y -3.5054,Z 86,A 176.9121,B 24.9145,C -2.1355,E1 24.8399,E2 267.9978} C_DIS
LIN {X -85.2858,Y -0.5852,Z 86,A 174.7845,B 24.9143,C -2.1373,E1 24.8398,E2 270.1341} C_DIS
LIN {X -85.2346,Y 3.0623,Z 86,A 172.1612,B 24.9141,C -2.1404,E1 24.84,E2 272.7657} C_DIS
LIN {X -84.9167,Y 7.9542,Z 86,A 168.7846,B 24.9134,C -2.1487,E1 24.8407,E2 276.1427} C_DIS
LIN {X -84.4928,Y 11.6279,Z 86,A 166.3777,B 24.9126,C -2.1587,E1 24.8415,E2 278.5401} C_DIS
LIN {X -83.6106,Y 16.837,Z 86,A 163.0035,B 24.9113,C -2.1748,E1 24.8432,E2 281.8961} C_DIS
LIN {X -82.9938,Y 19.6561,Z 86,A 160.9317,B 24.9111,C -2.1773,E1 24.8445,E2 283.9741} C_DIS
LIN {X -81.452,Y 25.2921,Z 86,A 157.5518,B 24.9089,C -2.2044,E1 24.847,E2 287.3088} C_DIS
LIN {X -80.2272,Y 28.9429,Z 86,A 154.1489,B 24.91,C -2.1901,E1 24.8501,E2 290.7652} C_DIS
LIN {X -78.709,Y 32.8493,Z 86,A 151.0605,B 24.91,C -2.1913,E1 24.8534,E2 293.868} C_DIS
LIN {X -77.4017,Y 35.8206,Z 86,A 149.3981,B 24.9082,C -2.2118,E1 24.8553,E2 295.4904} C_DIS
LIN {X -75.3176,Y 40.0183,Z 86,A 146.5097,B 24.9069,C -2.2282,E1 24.8589,E2 298.3553} C_DIS
LIN {X -74.2107,Y 42.0376,Z 86,A 144.7756,B 24.9069,C -2.2275,E1 24.8612,E2 300.1002} C_DIS
LIN {X -72.8212,Y 44.3981,Z 86,A 142.362,B 24.9078,C -2.2171,E1 24.8648,E2 302.551} C_DIS
LIN {X -70.331,Y 48.2486,Z 86,A 139.5577,B 24.9065,C -2.2331,E1 24.8691,E2 305.3311} C_DIS
LIN {X -67.6079,Y 51.9932,Z 86,A 136.0364,B 24.9067,C -2.2302,E1 24.875,E2 308.8762} C_DIS
LIN {X -65.5273,Y 54.5921,Z 86,A 134.3086,B 24.905,C -2.25,E1 24.878,E2 310.5649} C_DIS
LIN {X -62.64,Y 57.8815,Z 86,A 131.3108,B 24.9045,C -2.2558,E1 24.8836,E2 313.5623} C_DIS
LIN {X -60.0705,Y 60.5439,Z 86,A 128.5517,B 24.9047,C -2.2542,E1 24.8891,E2 316.3369} C_DIS
LIN {X -56.8442,Y 63.5834,Z 86,A 125.5741,B 24.9041,C -2.261,E1 24.8952,E2 319.3101} C_DIS
LIN {X -53.3562,Y 66.5389,Z 86,A 122.1504,B 24.9044,C -2.2579,E1 24.9026,E2 322.7543} C_DIS
LIN {X -50.4995,Y 68.7308,Z 86,A 120.7801,B 24.9014,C -2.2923,E1 24.9055,E2 324.0475} C_DIS
LIN {X -47.2058,Y 71.0338,Z 86,A 117.7163,B 24.9018,C -2.2873,E1 24.9126,E2 327.1336} C_DIS
LIN {X -45.0676,Y 72.4089,Z 86,A 115.4565,B 24.9029,C -2.2749,E1 24.9181,E2 329.43} C_DIS
LIN {X -41.2797,Y 74.6339,Z 86,A 113.0788,B 24.9011,C -2.2963,E1 24.9237,E2 331.7638} C_DIS
LIN {X -38.2433,Y 76.2347,Z 86,A 109.8713,B 24.9029,C -2.2745,E1 24.9319,E2 335.032} C_DIS
LIN {X -34.5131,Y 77.9947,Z 86,A 107.9225,B 24.9006,C -2.302,E1 24.9367,E2 336.92} C_DIS
LIN {X -31.7782,Y 79.1481,Z 86,A 105.4834,B 24.9014,C -2.292,E1 24.943,E2 339.3883} C_DIS
LIN {X -26.7179,Y 80.9969,Z 86,A 102.4491,B 24.8996,C -2.3134,E1 24.9509,E2 342.3776} C_DIS
LIN {X -23.2759,Y 82.0509,Z 86,A 99.9639,B 24.8996,C -2.3141,E1 24.9576,E2 344.8654} C_DIS
LIN {X -20.446,Y 82.8017,Z 86,A 97.8295,B 24.8998,C -2.3111,E1 24.9634,E2 347.0099} C_DIS
LIN {X -16.6371,Y 83.6514,Z 86,A 95.4207,B 24.899,C -2.3196,E1 24.9699,E2 349.4014} C_DIS
LIN {X -13.9481,Y 84.1402,Z 86,A 93.3706,B 24.8995,C -2.3147,E1 24.9756,E2 351.4654} C_DIS
LIN {X -8.6391,Y 84.8501,Z 86,A 89.9439,B 24.8988,C -2.3219,E1 24.985,E2 354.8774} C_DIS
LIN {X -3.8787,Y 85.2004,Z 86,A 86.74,B 24.8988,C -2.3233,E1 24.994,E2 358.0791} C_DIS
LIN {X 1.9869,Y 85.2663,Z 86,A 83.1066,B 24.8978,C -2.3334,E1 25.004,E2 361.6885} C_DIS
LIN {X 7.1389,Y 84.9898,Z 86,A 78.776,B 24.9001,C -2.3071,E1 25.0163,E2 366.0797} C_DIS
LIN {X 12.7239,Y 84.3345,Z 86,A 75.3756,B 24.8992,C -2.3178,E1 25.0256,E2 369.452} C_DIS
LIN {X 16.208,Y 83.7342,Z 86,A 72.9613,B 24.8994,C -2.3157,E1 25.0322,E2 371.8687} C_DIS
LIN {X 19.4304,Y 83.0459,Z 86,A 70.8698,B 24.8992,C -2.3183,E1 25.0379,E2 373.951} C_DIS
LIN {X 22.4504,Y 82.2808,Z 86,A 68.6711,B 24.8996,C -2.3138,E1 25.0439,E2 376.1571} C_DIS
LIN {X 25.7449,Y 81.3116,Z 86,A 66.0644,B 24.9005,C -2.3027,E1 25.0509,E2 378.7854} C_DIS
LIN {X 29.5632,Y 80.0016,Z 86,A 63.17,B 24.9012,C -2.2946,E1 25.0585,E2 381.693} C_DIS
LIN {X 32.6493,Y 78.7925,Z 86,A 61.5179,B 24.8999,C -2.3103,E1 25.0627,E2 383.3042} C_DIS
LIN {X 36.0115,Y 77.3129,Z 86,A 58.0902,B 24.9027,C -2.2774,E1 25.0716,E2 386.8009} C_DIS
LIN {X 40.1514,Y 75.2475,Z 86,A 56.1664,B 24.8998,C -2.3106,E1 25.0761,E2 388.6408} C_DIS
LIN {X 45.5927,Y 72.0808,Z 86,A 51.8844,B 24.9005,C -2.3028,E1 25.0864,E2 392.9283} C_DIS
LIN {X 47.6768,Y 70.7182,Z 86,A 50.0425,B 24.9012,C -2.2947,E1 25.0907,E2 394.7831} C_DIS
LIN {X 51.9947,Y 67.6067,Z 86,A 46.2167,B 24.9024,C -2.2805,E1 25.0994,E2 398.629} C_DIS
LIN {X 54.9204,Y 65.2543,Z 86,A 44.0026,B 24.902,C -2.2857,E1 25.1041,E2 400.8224} C_DIS
LIN {X 57.2369,Y 63.2318,Z 86,A 41.9142,B 24.9024,C -2.2809,E1 25.1085,E2 402.9138} C_DIS
LIN {X 59.4878,Y 61.1186,Z 86,A 39.5227,B 24.9036,C -2.2663,E1 25.1133,E2 405.3299} C_DIS
LIN {X 63.1728,Y 57.3012,Z 86,A 36.0011,B 24.9042,C -2.2599,E1 25.1201,E2 408.8513} C_DIS
LIN {X 65.6577,Y 54.4352,Z 86,A 33.8185,B 24.9037,C -2.266,E1 25.124,E2 411.0095} C_DIS
LIN {X 68.7165,Y 50.5191,Z 86,A 30.4814,B 24.9044,C -2.258,E1 25.1296,E2 414.3497} C_DIS
LIN {X 70.3346,Y 48.2434,Z 86,A 28.4728,B 24.9051,C -2.2489,E1 25.1329,E2 416.37} C_DIS
LIN {X 73.1557,Y 43.8478,Z 86,A 25.0088,B 24.9058,C -2.2412,E1 25.138,E2 419.8345} C_DIS
LIN {X 74.8969,Y 40.7993,Z 86,A 21.8581,B 24.9085,C -2.2088,E1 25.1423,E2 423.0454} C_DIS
LIN {X 76.911,Y 36.8618,Z 86,A 19.9188,B 24.9063,C -2.2347,E1 25.1446,E2 424.9131} C_DIS
LIN {X 77.9139,Y 34.6941,Z 86,A 17.1179,B 24.91,C -2.1904,E1 25.1479,E2 427.8032} C_DIS
LIN {X 79.8216,Y 30.0441,Z 86,A 15.2459,B 24.9067,C -2.2307,E1 25.1497,E2 429.5697} C_DIS
LIN {X 80.6729,Y 27.6804,Z 86,A 13.3746,B 24.9076,C -2.2196,E1 25.1514,E2 431.4569} C_DIS
LIN {X 81.4724,Y 25.2261,Z 86,A 11.4967,B 24.9084,C -2.2096,E1 25.153,E2 433.3477} C_DIS
LIN {X 82.3703,Y 22.1193,Z 86,A 9.3043,B 24.909,C -2.2023,E1 25.1547,E2 435.5447} C_DIS
LIN {X 83.1653,Y 18.9139,Z 86,A 6.3328,B 24.9117,C -2.1703,E1 25.1566,E2 438.5745} C_DIS
LIN {X 83.954,Y 15.0281,Z 86,A 3.9567,B 24.9115,C -2.1716,E1 25.1578,E2 440.9336} C_DIS
LIN {X 84.7481,Y 9.5902,Z 86,A 0.6912,B 24.9113,C -2.1744,E1 25.159,E2 444.1733} C_DIS
LIN {X 85.1136,Y 5.455,Z 86,A -2.0458,B 24.9119,C -2.1673,E1 25.1595,E2 446.9107} C_DIS
LIN {X 85.2677,Y 1.844,Z 86,A -4.6984,B 24.9131,C -2.152,E1 25.1598,E2 449.5838} C_DIS
LIN {X 85.2482,Y -2.6188,Z 86,A -7.9019,B 24.9145,C -2.1355,E1 25.1596,E2 452.8071} C_DIS
LIN {X 85.088,Y -5.8441,Z 86,A -10.2184,B 24.9154,C -2.1236,E1 25.1591,E2 455.138} C_DIS
LIN {X 84.7467,Y -9.6023,Z 86,A -11.9624,B 24.9139,C -2.1422,E1 25.1586,E2 456.8279} C_DIS
LIN {X 84.3881,Y -12.3649,Z 86,A -14.4449,B 24.9161,C -2.1155,E1 25.1576,E2 459.3586} C_DIS
LIN {X 83.847,Y -15.6216,Z 86,A -16.1807,B 24.9153,C -2.1247,E1 25.1568,E2 461.0625} C_DIS
LIN {X 82.5727,Y -21.3511,Z 86,A -20.2528,B 24.9167,C -2.1079,E1 25.1542,E2 465.1507} C_DIS
LIN {X 81.0374,Y -26.5927,Z 86,A -23.4345,B 24.9163,C -2.113,E1 25.1516,E2 468.3023} C_DIS
LIN {X 79.3896,Y -31.1674,Z 86,A -26.8754,B 24.9175,C -2.097,E1 25.1483,E2 471.7617} C_DIS
LIN {X 78.1915,Y -34.0616,Z 86,A -28.9985,B 24.9181,C -2.09,E1 25.146,E2 473.8897} C_DIS
LIN {X 76.2498,Y -38.2128,Z 86,A -32.1465,B 24.919,C -2.0784,E1 25.1422,E2 477.048} C_DIS
LIN {X 73.6123,Y -43.0753,Z 86,A -35.5256,B 24.919,C -2.079,E1 25.1377,E2 480.4081} C_DIS
LIN {X 70.8242,Y -47.5203,Z 86,A -39.0058,B 24.9196,C -2.0706,E1 25.1325,E2 483.8908} C_DIS
LIN {X 68.8318,Y -50.3617,Z 86,A -41.8424,B 24.9214,C -2.0472,E1 25.1278,E2 486.7687} C_DIS
LIN {X 66.4088,Y -53.5161,Z 86,A -44.2933,B 24.9214,C -2.0475,E1 25.1236,E2 489.2074} C_DIS
LIN {X 64.4495,Y -55.8612,Z 86,A -46.2916,B 24.9217,C -2.0441,E1 25.12,E2 491.2048} C_DIS
LIN {X 62.345,Y -58.2006,Z 86,A -48.8553,B 24.9232,C -2.0238,E1 25.115,E2 493.805} C_DIS
LIN {X 58.0117,Y -62.52,Z 86,A -52.688,B 24.9232,C -2.0232,E1 25.1074,E2 497.6232} C_DIS
LIN {X 54.7899,Y -65.3629,Z 86,A -55.948,B 24.9247,C -2.0044,E1 25.1004,E2 500.9149} C_DIS
LIN {X 52.1005,Y -67.5252,Z 86,A -57.8822,B 24.9241,C -2.0121,E1 25.0962,E2 502.8239} C_DIS
LIN {X 48.1237,Y -70.4156,Z 86,A -60.6867,B 24.9234,C -2.0217,E1 25.0899,E2 505.5959} C_DIS
LIN {X 44.781,Y -72.5869,Z 86,A -63.7024,B 24.9246,C -2.0055,E1 25.0827,E2 508.6401} C_DIS
LIN {X 40.1469,Y -75.2499,Z 86,A -66.985,B 24.9243,C -2.0091,E1 25.0748,E2 511.9044} C_DIS
LIN {X 35.5816,Y -77.513,Z 86,A -70.4372,B 24.9248,C -2.0027,E1 25.0661,E2 515.3627} C_DIS
LIN {X 30.8908,Y -79.4982,Z 86,A -73.7204,B 24.9248,C -2.0022,E1 25.0577,E2 518.6393} C_DIS
LIN {X 27.2451,Y -80.8196,Z 86,A -76.6853,B 24.926,C -1.9873,E1 25.0498,E2 521.6336} C_DIS
LIN {X 22.8394,Y -82.1743,Z 86,A -79.5274,B 24.9256,C -1.9919,E1 25.0422,E2 524.4598} C_DIS
LIN {X 20.9081,Y -82.6866,Z 86,A -81.9581,B 24.9283,C -1.9562,E1 25.0354,E2 526.9715} C_DIS
LIN {X 16.4992,Y -83.6781,Z 86,A -84.0692,B 24.9263,C -1.9825,E1 25.0298,E2 529.0174} C_DIS
LIN {X 11.3022,Y -84.5369,Z 86,A -87.6459,B 24.9266,C -1.9788,E1 25.0199,E2 532.5996} C_DIS
LIN {X 5.0835,Y -85.1376,Z 86,A -91.9232,B 24.9269,C -1.9742,E1 25.008,E2 536.8856} C_DIS
LIN {X 0.5378,Y -85.2804,Z 86,A -93.6627,B 24.9239,C -2.0145,E1 25.0035,E2 538.5288} C_DIS
Enddeposition()
LIN {X 0.5378,Y -85.2804,Z 86,A -93.6627,B 24.9239,C -2.0145,E1 25.0035,E2 538.5288} C_DIS
Startdeposition()
$VEL.CP = VEL_PRINT
LIN {X 0.8604,Y -84.3776,Z 86,A -93.0048,B 24.9217,C -2.0438,E1 25.0055,E2 537.8015} C_DIS
LIN {X 4.5186,Y -84.2603,Z 86,A -91.3231,B 24.9235,C -2.0195,E1 25.01,E2 536.1782} C_DIS
LIN {X 9.3897,Y -83.8583,Z 86,A -87.834,B 24.923,C -2.0265,E1 25.0197,E2 532.6744} C_DIS
LIN {X 12.5346,Y -83.4459,Z 86,A -85.6482,B 24.9228,C -2.029,E1 25.0258,E2 530.4847} C_DIS
LIN {X 16.7361,Y -82.7053,Z 86,A -82.1796,B 24.9212,C -2.0497,E1 25.0354,E2 526.971} C_DIS
LIN {X 20.2957,Y -81.9047,Z 86,A -80.4765,B 24.9229,C -2.0272,E1 25.0399,E2 525.3236} C_DIS
LIN {X 23.0574,Y -81.17,Z 86,A -77.9686,B 24.9214,C -2.0476,E1 25.0467,E2 522.7716} C_DIS
LIN {X 26.9343,Y -79.9672,Z 86,A -75.6677,B 24.9223,C -2.0362,E1 25.0528,E2 520.5021} C_DIS
LIN {X 30.6403,Y -78.6221,Z 86,A -72.4018,B 24.9205,C -2.0589,E1 25.0614,E2 517.1893} C_DIS
LIN {X 33.8524,Y -77.2932,Z 86,A -70.6119,B 24.9217,C -2.0438,E1 25.0659,E2 515.4396} C_DIS
LIN {X 39.1461,Y -74.7517,Z 86,A -66.7679,B 24.9215,C -2.0455,E1 25.0755,E2 511.6018} C_DIS
LIN {X 42.701,Y -72.7798,Z 86,A -62.9616,B 24.9185,C -2.0851,E1 25.0849,E2 507.7134} C_DIS
LIN {X 46.6345,Y -70.3241,Z 86,A -60.7454,B 24.9204,C -2.0601,E1 25.0899,E2 505.5634} C_DIS
LIN {X 50.3717,Y -67.6973,Z 86,A -57.7593,B 24.9202,C -2.0627,E1 25.0967,E2 502.5818} C_DIS
LIN {X 55.1412,Y -63.874,Z 86,A -53.5025,B 24.9192,C -2.0753,E1 25.1059,E2 498.3114} C_DIS
LIN {X 58.1265,Y -61.1679,Z 86,A -50.7355,B 24.9187,C -2.0827,E1 25.1116,E2 495.538} C_DIS
LIN {X 60.9841,Y -58.3202,Z 86,A -47.8642,B 24.9178,C -2.0938,E1 25.1172,E2 492.6527} C_DIS
LIN {X 63.7782,Y -55.2508,Z 86,A -44.3625,B 24.9154,C -2.1242,E1 25.1238,E2 489.0952} C_DIS
LIN {X 66.7024,Y -51.6822,Z 86,A -42.5614,B 24.9183,C -2.0874,E1 25.1268,E2 487.3893} C_DIS
LIN {X 69.6119,Y -47.6928,Z 86,A -38.8156,B 24.9165,C -2.1097,E1 25.1329,E2 483.609} C_DIS
LIN {X 71.0585,Y -45.5072,Z 86,A -36.8516,B 24.9156,C -2.121,E1 25.1359,E2 481.6283} C_DIS
LIN {X 73.0449,Y -42.2458,Z 86,A -34.055,B 24.9145,C -2.1353,E1 25.1399,E2 478.8122} C_DIS
LIN {X 75.1698,Y -38.3368,Z 86,A -31.7199,B 24.9156,C -2.1209,E1 25.1428,E2 476.5236} C_DIS
LIN {X 76.6326,Y -35.3235,Z 86,A -29.1369,B 24.9143,C -2.1381,E1 25.146,E2 473.9138} C_DIS
LIN {X 78.1103,Y -31.9218,Z 86,A -26.9516,B 24.9146,C -2.1344,E1 25.1483,E2 471.7491} C_DIS
LIN {X 79.5947,Y -28.016,Z 86,A -23.9319,B 24.9134,C -2.1493,E1 25.1513,E2 468.7111} C_DIS
LIN {X 80.9568,Y -23.796,Z 86,A -20.4569,B 24.9113,C -2.1746,E1 25.1542,E2 465.1962} C_DIS
LIN {X 82.574,Y -17.3753,Z 86,A -16.1883,B 24.9108,C -2.181,E1 25.1569,E2 460.9373} C_DIS
LIN {X 83.3666,Y -13.0474,Z 86,A -13.561,B 24.911,C -2.1782,E1 25.1581,E2 458.332} C_DIS
LIN {X 83.783,Y -10.033,Z 86,A -11.5878,B 24.9107,C -2.1816,E1 25.1588,E2 456.3624} C_DIS
LIN {X 84.178,Y -5.8556,Z 86,A -7.7796,B 24.9072,C -2.2236,E1 25.1596,E2 452.4776} C_DIS
LIN {X 84.3672,Y -1.5447,Z 86,A -5.7407,B 24.909,C -2.2024,E1 25.1598,E2 450.5009} C_DIS
LIN {X 84.351,Y 2.2802,Z 86,A -3.0946,B 24.9082,C -2.2123,E1 25.1597,E2 447.847} C_DIS
LIN {X 84.1535,Y 6.1899,Z 86,A -0.1139,B 24.9066,C -2.2318,E1 25.1591,E2 444.8381} C_DIS
LIN {X 83.0906,Y 14.704,Z 86,A 5.8411,B 24.9047,C -2.2544,E1 25.1568,E2 438.8649} C_DIS
LIN {X 82.439,Y 18.0004,Z 86,A 7.4625,B 24.906,C -2.2389,E1 25.1558,E2 437.2894} C_DIS
LIN {X 81.7601,Y 20.8691,Z 86,A 9.4972,B 24.9054,C -2.2462,E1 25.1545,E2 435.2494} C_DIS
LIN {X 80.8939,Y 24.008,Z 86,A 11.7545,B 24.9047,C -2.2544,E1 25.1527,E2 432.9857} C_DIS
LIN {X 79.9343,Y 27.0318,Z 86,A 14.1922,B 24.9033,C -2.2704,E1 25.1506,E2 430.524} C_DIS
LIN {X 78.93,Y 29.8372,Z 86,A 16.4028,B 24.9022,C -2.2826,E1 25.1484,E2 428.2967} C_DIS
LIN {X 77.7225,Y 32.8546,Z 86,A 18.1483,B 24.903,C -2.2733,E1 25.1465,E2 426.5827} C_DIS
LIN {X 76.2304,Y 36.1841,Z 86,A 21.483,B 24.8999,C -2.3093,E1 25.1425,E2 423.1811} C_DIS
LIN {X 74.1612,Y 40.2532,Z 86,A 23.6415,B 24.902,C -2.2859,E1 25.1397,E2 421.0891} C_DIS
LIN {X 72.3776,Y 43.3815,Z 86,A 27.0102,B 24.8987,C -2.3234,E1 25.1348,E2 417.6491} C_DIS
LIN {X 69.9114,Y 47.2505,Z 86,A 29.1002,B 24.901,C -2.297,E1 25.1317,E2 415.632} C_DIS
LIN {X 68.5746,Y 49.1708,Z 86,A 31.7719,B 24.8975,C -2.3371,E1 25.1272,E2 412.8783} C_DIS
LIN {X 65.6029,Y 53.0704,Z 86,A 34.027,B 24.9,C -2.3092,E1 25.1234,E2 410.6999} C_DIS
LIN {X 64.2123,Y 54.7447,Z 86,A 36.0561,B 24.8981,C -2.3308,E1 25.1197,E2 408.6288} C_DIS
LIN {X 61.9918,Y 57.2476,Z 86,A 37.5519,B 24.8999,C -2.3102,E1 25.1169,E2 407.1883} C_DIS
LIN {X 59.0267,Y 60.3009,Z 86,A 40.703,B 24.8986,C -2.3249,E1 25.1107,E2 404.0159} C_DIS
LIN {X 56.3447,Y 62.8131,Z 86,A 43.0689,B 24.8986,C -2.3257,E1 25.1059,E2 401.6577} C_DIS
LIN {X 54.061,Y 64.7892,Z 86,A 44.9877,B 24.8986,C -2.3254,E1 25.1018,E2 399.7472} C_DIS
LIN {X 51.7729,Y 66.6325,Z 86,A 47.4481,B 24.8969,C -2.3441,E1 25.0963,E2 397.2517} C_DIS
LIN {X 47.5462,Y 69.7112,Z 86,A 50.7063,B 24.8972,C -2.3406,E1 25.089,E2 394.0131} C_DIS
LIN {X 43.7237,Y 72.1697,Z 86,A 54.2757,B 24.8954,C -2.3609,E1 25.0804,E2 390.407} C_DIS
LIN {X 39.4024,Y 74.6168,Z 86,A 58.3436,B 24.893,C -2.3878,E1 25.0703,E2 386.2867} C_DIS
LIN {X 34.5347,Y 76.9908,Z 86,A 60.7912,B 24.8961,C -2.3526,E1 25.0643,E2 383.9288} C_DIS
LIN {X 32.2555,Y 77.9744,Z 86,A 62.5511,B 24.8958,C -2.3567,E1 25.0597,E2 382.1632} C_DIS
LIN {X 28.5839,Y 79.3932,Z 86,A 64.8831,B 24.8965,C -2.3486,E1 25.0537,E2 379.8556} C_DIS
LIN {X 25.2526,Y 80.5145,Z 86,A 67.5546,B 24.8955,C -2.3594,E1 25.0466,E2 377.1635} C_DIS
LIN {X 22.0684,Y 81.4444,Z 86,A 69.7899,B 24.8955,C -2.3604,E1 25.0406,E2 374.9296} C_DIS
LIN {X 18.9689,Y 82.2216,Z 86,A 71.8724,B 24.8955,C -2.3589,E1 25.0349,E2 372.8537} C_DIS
LIN {X 15.9614,Y 82.8579,Z 86,A 73.8176,B 24.8959,C -2.3554,E1 25.0296,E2 370.919} C_DIS
LIN {X 12.3541,Y 83.4735,Z 86,A 77.5207,B 24.8925,C -2.3939,E1 25.0192,E2 367.1282} C_DIS
LIN {X 7.6918,Y 84.03,Z 86,A 79.7477,B 24.8951,C -2.3646,E1 25.0132,E2 364.9722} C_DIS
LIN {X 2.5138,Y 84.3439,Z 86,A 83.0798,B 24.8956,C -2.3587,E1 25.0039,E2 361.6553} C_DIS
LIN {X -2.5268,Y 84.3435,Z 86,A 86.6124,B 24.8954,C -2.3612,E1 24.9941,E2 358.1166} C_DIS
LIN {X -5.1952,Y 84.2226,Z 86,A 88.6113,B 24.895,C -2.3661,E1 24.9884,E2 356.1055} C_DIS
LIN {X -9.0801,Y 83.8919,Z 86,A 91.5715,B 24.8942,C -2.3741,E1 24.9802,E2 353.1245} C_DIS
LIN {X -13.8261,Y 83.2409,Z 86,A 94.1693,B 24.8962,C -2.3524,E1 24.9731,E2 350.5761} C_DIS
LIN {X -16.73,Y 82.7065,Z 86,A 96.0409,B 24.8966,C -2.3469,E1 24.968,E2 348.7156} C_DIS
LIN {X -19.1989,Y 82.1684,Z 86,A 98.1571,B 24.8957,C -2.3572,E1 24.9622,E2 346.5723} C_DIS
LIN {X -22.526,Y 81.3205,Z 86,A 101.2619,B 24.8939,C -2.3777,E1 24.9537,E2 343.4139} C_DIS
LIN {X -26.504,Y 80.1123,Z 86,A 103.8784,B 24.8948,C -2.3682,E1 24.9468,E2 340.8152} C_DIS
LIN {X -29.7333,Y 78.9694,Z 86,A 106.0123,B 24.8955,C -2.3596,E1 24.9412,E2 338.6975} C_DIS
LIN {X -33.5048,Y 77.4447,Z 86,A 108.7332,B 24.896,C -2.3544,E1 24.9343,E2 335.9826} C_DIS
LIN {X -37.8113,Y 75.4364,Z 86,A 112.019,B 24.8963,C -2.351,E1 24.926,E2 332.6962} C_DIS
LIN {X -41.6311,Y 73.3981,Z 86,A 114.3651,B 24.8982,C -2.3289,E1 24.9204,E2 330.396} C_DIS
LIN {X -45.75,Y 70.9026,Z 86,A 118.7426,B 24.896,C -2.3546,E1 24.9099,E2 325.9434} C_DIS
LIN {X -49.4097,Y 68.4041,Z 86,A 120.841,B 24.8988,C -2.3225,E1 24.9052,E2 323.9143} C_DIS
LIN {X -52.777,Y 65.8407,Z 86,A 124.4275,B 24.8976,C -2.3367,E1 24.8973,E2 320.2809} C_DIS
LIN {X -55.5525,Y 63.5148,Z 86,A 126.2818,B 24.8995,C -2.3141,E1 24.8934,E2 318.4733} C_DIS
LIN {X -58.0419,Y 61.249,Z 86,A 128.2237,B 24.9008,C -2.2992,E1 24.8895,E2 316.5589} C_DIS
LIN {X -60.8682,Y 58.4405,Z 86,A 131.8541,B 24.8991,C -2.3186,E1 24.8823,E2 312.8668} C_DIS
LIN {X -63.2603,Y 55.8439,Z 86,A 133.6857,B 24.901,C -2.2967,E1 24.879,E2 311.0792} C_DIS
LIN {X -65.4655,Y 53.24,Z 86,A 137.3535,B 24.8983,C -2.3286,E1 24.8724,E2 307.318} C_DIS
LIN {X -69.0232,Y 48.5409,Z 86,A 140.0633,B 24.9023,C -2.2815,E1 24.8681,E2 304.7076} C_DIS
LIN {X -70.5221,Y 46.3342,Z 86,A 142.5959,B 24.901,C -2.2966,E1 24.8642,E2 302.1263} C_DIS
LIN {X -72.6129,Y 42.9834,Z 86,A 144.4873,B 24.9036,C -2.267,E1 24.8615,E2 300.2957} C_DIS
LIN {X -74.3873,Y 39.8364,Z 86,A 147.8178,B 24.9021,C -2.2842,E1 24.857,E2 296.9067} C_DIS
LIN {X -76.2413,Y 36.1614,Z 86,A 149.9125,B 24.9045,C -2.2565,E1 24.8545,E2 294.8666} C_DIS
LIN {X -78.0515,Y 32.0662,Z 86,A 152.9332,B 24.9053,C -2.2468,E1 24.8512,E2 291.8524} C_DIS
LIN {X -80.46,Y 25.4283,Z 86,A 157.6498,B 24.9067,C -2.2299,E1 24.8469,E2 287.1494} C_DIS
LIN {X -81.9923,Y 19.9367,Z 86,A 161.6562,B 24.9074,C -2.2214,E1 24.844,E2 283.1399} C_DIS
LIN {X -83.238,Y 13.8433,Z 86,A 166.1988,B 24.9078,C -2.2167,E1 24.8416,E2 278.5816} C_DIS
LIN {X -83.7698,Y 10.1458,Z 86,A 168.4888,B 24.9091,C -2.2019,E1 24.8407,E2 276.3134} C_DIS
LIN {X -84.1394,Y 6.3939,Z 86,A 170.7565,B 24.9104,C -2.1857,E1 24.8402,E2 274.0706} C_DIS
LIN {X -84.3114,Y 3.4379,Z 86,A 172.9699,B 24.9104,C -2.1848,E1 24.8399,E2 271.8461} C_DIS
LIN {X -84.3797,Y 0.3739,Z 86,A 175.6694,B 24.9096,C -2.1952,E1 24.8399,E2 269.1056} C_DIS
LIN {X -84.3283,Y -3.0144,Z 86,A 177.6556,B 24.9109,C -2.1792,E1 24.8399,E2 267.1458} C_DIS
LIN {X -84.1222,Y -6.6084,Z 86,A 179.8268,B 24.9122,C -2.1639,E1 24.8404,E2 264.9977} C_DIS
LIN {X -83.7382,Y -10.4022,Z 86,A -177.4155,B 24.9125,C -2.1604,E1 24.8412,E2 262.232} C_DIS
LIN {X -83.2013,Y -14.0628,Z 86,A -175.1614,B 24.9137,C -2.1455,E1 24.8422,E2 260.0001} C_DIS
LIN {X -82.4902,Y -17.7659,Z 86,A -171.7818,B 24.9125,C -2.1602,E1 24.8441,E2 256.5655} C_DIS
LIN {X -81.6897,Y -21.1426,Z 86,A -170.0007,B 24.9143,C -2.1371,E1 24.8453,E2 254.8291} C_DIS
LIN {X -80.9922,Y -23.6766,Z 86,A -167.807,B 24.9139,C -2.143,E1 24.8471,E2 252.6085} C_DIS
LIN {X -79.4569,Y -28.4086,Z 86,A -164.3254,B 24.9144,C -2.136,E1 24.8502,E2 249.124} C_DIS
LIN {X -77.7787,Y -32.7212,Z 86,A -161.7202,B 24.9163,C -2.112,E1 24.8529,E2 246.5615} C_DIS
LIN {X -76.7881,Y -34.9844,Z 86,A -160.003,B 24.9166,C -2.1084,E1 24.8549,E2 244.8435} C_DIS
LIN {X -75.5007,Y -37.6816,Z 86,A -157.8827,B 24.9169,C -2.1053,E1 24.8575,E2 242.7191} C_DIS
LIN {X -73.2032,Y -41.9703,Z 86,A -154.1292,B 24.9166,C -2.109,E1 24.8626,E2 238.9369} C_DIS
LIN {X -70.6184,Y -46.1881,Z 86,A -151.3851,B 24.9186,C -2.083,E1 24.8666,E2 236.2409} C_DIS
LIN {X -69.1394,Y -48.3728,Z 86,A -148.7466,B 24.9171,C -2.1026,E1 24.8709,E2 233.5429} C_DIS
LIN {X -66.9463,Y -51.3656,Z 86,A -146.8912,B 24.9191,C -2.0776,E1 24.874,E2 231.7381} C_DIS
LIN {X -64.5739,Y -54.32,Z 86,A -143.218,B 24.917,C -2.1032,E1 24.8807,E2 227.987} C_DIS
LIN {X -61.277,Y -58.0122,Z 86,A -140.8943,B 24.92,C -2.0659,E1 24.885,E2 225.742} C_DIS
LIN {X -59.1435,Y -60.1855,Z 86,A -138.585,B 24.9198,C -2.0685,E1 24.8896,E2 223.4167} C_DIS
LIN {X -56.1412,Y -62.9952,Z 86,A -136.0548,B 24.9208,C -2.0554,E1 24.8947,E2 220.9074} C_DIS
LIN {X -54.3595,Y -64.5405,Z 86,A -134.0044,B 24.92,C -2.0654,E1 24.8992,E2 218.8254} C_DIS
LIN {X -49.3499,Y -68.4468,Z 86,A -130.0159,B 24.9213,C -2.0484,E1 24.908,E2 214.8631} C_DIS
LIN {X -44.2079,Y -71.8754,Z 86,A -125.7594,B 24.9217,C -2.0436,E1 24.918,E2 210.6042} C_DIS
LIN {X -37.92,Y -75.3822,Z 86,A -120.9335,B 24.9223,C -2.0352,E1 24.9298,E2 205.7846} C_DIS
LIN {X -34.9437,Y -76.8065,Z 86,A -118.6663,B 24.9225,C -2.0334,E1 24.9355,E2 203.5158} C_DIS
LIN {X -31.2951,Y -78.3648,Z 86,A -115.5126,B 24.9216,C -2.0445,E1 24.9438,E2 200.3287} C_DIS
LIN {X -28.2914,Y -79.4981,Z 86,A -113.9772,B 24.9232,C -2.0232,E1 24.9477,E2 198.8409} C_DIS
LIN {X -24.5961,Y -80.7181,Z 86,A -111.1333,B 24.9229,C -2.0273,E1 24.9553,E2 195.9823} C_DIS
LIN {X -21.5063,Y -81.5963,Z 86,A -108.9926,B 24.9231,C -2.0247,E1 24.961,E2 193.8444} C_DIS
LIN {X -18.9416,Y -82.2279,Z 86,A -106.7371,B 24.9221,C -2.0379,E1 24.9673,E2 191.5544} C_DIS
LIN {X -15.4509,Y -82.9562,Z 86,A -103.629,B 24.9206,C -2.0583,E1 24.976,E2 188.3948} C_DIS
LIN {X -10.2361,Y -83.7592,Z 86,A -101.45,B 24.9239,C -2.0141,E1 24.9817,E2 186.3191} C_DIS
LIN {X -7.0613,Y -84.0853,Z 86,A -98.8868,B 24.923,C -2.0262,E1 24.9889,E2 183.7259} C_DIS
LIN {X -2.9528,Y -84.3286,Z 86,A -95.8846,B 24.9225,C -2.0329,E1 24.9973,E2 180.7071} C_DIS
LIN {X 0.533,Y -84.3793,Z 86,A -94.4452,B 24.9247,C -2.0045,E1 25.0012,E2 179.3349} C_DIS
Enddeposition()
LIN {X 0.533,Y -84.3793,Z 86,A -94.4452,B 24.9247,C -2.0045,E1 25.0012,E2 179.3349} C_DIS
Startdeposition()
$VEL.CP = VEL_PRINT
LIN {X -0.7285,Y -83.4713,Z 86,A -96.3891,B 24.9259,C -1.9876,E1 24.9956,E2 181.319} C_DIS
LIN {X -4.2032,Y -83.3693,Z 86,A -98.8742,B 24.9262,C -1.9845,E1 24.9887,E2 183.8122} C_DIS
LIN {X -7.918,Y -83.0982,Z 86,A -100.5928,B 24.9243,C -2.0096,E1 24.9841,E2 185.472} C_DIS
LIN {X -11.0373,Y -82.7419,Z 86,A -103.6833,B 24.9263,C -1.9823,E1 24.9753,E2 188.6297} C_DIS
LIN {X -15.031,Y -82.1102,Z 86,A -105.401,B 24.9239,C -2.0143,E1 24.9708,E2 190.273} C_DIS
LIN {X -18.2227,Y -81.4621,Z 86,A -107.9278,B 24.9245,C -2.0067,E1 24.9638,E2 192.821} C_DIS
LIN {X -21.2751,Y -80.7191,Z 86,A -110.0855,B 24.9245,C -2.0078,E1 24.958,E2 194.979} C_DIS
LIN {X -24.2174,Y -79.8856,Z 86,A -112.4949,B 24.925,C -2.0002,E1 24.9515,E2 197.4105} C_DIS
LIN {X -27.4446,Y -78.8339,Z 86,A -114.9723,B 24.9252,C -1.9979,E1 24.9449,E2 199.8982} C_DIS
LIN {X -31.0563,Y -77.4833,Z 86,A -117.659,B 24.9251,C -1.9993,E1 24.9379,E2 202.5875} C_DIS
LIN {X -35.7303,Y -75.4421,Z 86,A -120.6889,B 24.9237,C -2.0166,E1 24.9303,E2 205.5835} C_DIS
LIN {X -38.371,Y -74.1336,Z 86,A -123.4644,B 24.9252,C -1.9978,E1 24.9233,E2 208.4113} C_DIS
LIN {X -41.8411,Y -72.2312,Z 86,A -125.483,B 24.9234,C -2.0213,E1 24.9185,E2 210.3801} C_DIS
LIN {X -47.2727,Y -68.8,Z 86,A -129.626,B 24.9223,C -2.0356,E1 24.9088,E2 214.5023} C_DIS
LIN {X -51.322,Y -65.8333,Z 86,A -133.9868,B 24.9238,C -2.016,E1 24.899,E2 218.9254} C_DIS
LIN {X -54.1921,Y -63.4915,Z 86,A -135.3117,B 24.9208,C -2.0547,E1 24.8963,E2 220.1631} C_DIS
LIN {X -55.7336,Y -62.1427,Z 86,A -137.3386,B 24.922,C -2.0401,E1 24.892,E2 222.233} C_DIS
LIN {X -58.3018,Y -59.7418,Z 86,A -139.7438,B 24.9216,C -2.0452,E1 24.8871,E2 224.6359} C_DIS
LIN {X -60.5438,Y -57.4678,Z 86,A -142.6392,B 24.9227,C -2.0306,E1 24.8815,E2 227.5786} C_DIS
LIN {X -63.1485,Y -54.5922,Z 86,A -144.8979,B 24.9214,C -2.0477,E1 24.8774,E2 229.8069} C_DIS
LIN {X -65.6619,Y -51.5415,Z 86,A -147.4432,B 24.9205,C -2.0586,E1 24.8729,E2 232.3379} C_DIS
LIN {X -68.7619,Y -47.3276,Z 86,A -150.7048,B 24.9191,C -2.0764,E1 24.8677,E2 235.573} C_DIS
LIN {X -70.0406,Y -45.4138,Z 86,A -153.093,B 24.9205,C -2.0586,E1 24.8639,E2 238.0158} C_DIS
LIN {X -71.8235,Y -42.5363,Z 86,A -154.5447,B 24.9182,C -2.0882,E1 24.8619,E2 239.4043} C_DIS
LIN {X -73.9494,Y -38.723,Z 86,A -157.2819,B 24.917,C -2.1033,E1 24.8583,E2 242.1199} C_DIS
LIN {X -75.7361,Y -35.0999,Z 86,A -160.6463,B 24.9177,C -2.0949,E1 24.8541,E2 245.5224} C_DIS
LIN {X -76.9821,Y -32.2759,Z 86,A -162.7907,B 24.9173,C -2.1003,E1 24.8517,E2 247.6659} C_DIS
LIN {X -78.6057,Y -28.0949,Z 86,A -166.7211,B 24.9183,C -2.0867,E1 24.8479,E2 251.651} C_DIS
LIN {X -79.917,Y -24.1116,Z 86,A -168.8739,B 24.9162,C -2.1144,E1 24.8461,E2 253.7499} C_DIS
LIN {X -81.1598,Y -19.5182,Z 86,A -172.1506,B 24.9154,C -2.1241,E1 24.8438,E2 257.0227} C_DIS
LIN {X -81.9141,Y -16.0635,Z 86,A -174.5839,B 24.9148,C -2.1314,E1 24.8425,E2 259.453} C_DIS
LIN {X -82.5112,Y -12.6438,Z 86,A -176.8656,B 24.914,C -2.1415,E1 24.8414,E2 261.7241} C_DIS
LIN {X -83.0923,Y -7.9824,Z 86,A -179.839,B 24.9126,C -2.1582,E1 24.8405,E2 264.6752} C_DIS
LIN {X -83.2838,Y -5.6353,Z 86,A 178.3251,B 24.9126,C -2.1575,E1 24.8401,E2 266.5238} C_DIS
LIN {X -83.4361,Y -2.5211,Z 86,A 175.6714,B 24.9132,C -2.1508,E1 24.8398,E2 269.2095} C_DIS
LIN {X -83.4567,Y 1.7173,Z 86,A 173.2095,B 24.9115,C -2.1718,E1 24.8398,E2 271.6361} C_DIS
LIN {X -83.3271,Y 4.9495,Z 86,A 170.8361,B 24.9113,C -2.1749,E1 24.8402,E2 274.0164} C_DIS
LIN {X -83.0292,Y 8.6086,Z 86,A 168.4429,B 24.9103,C -2.1863,E1 24.8408,E2 276.3969} C_DIS
LIN {X -82.7768,Y 10.7679,Z 86,A 166.3003,B 24.9114,C -2.174,E1 24.8416,E2 278.5816} C_DIS
LIN {X -82.2794,Y 14.0765,Z 86,A 164.3753,B 24.91,C -2.191,E1 24.8424,E2 280.4774} C_DIS
LIN {X -81.3803,Y 18.5806,Z 86,A 161.6159,B 24.9083,C -2.2113,E1 24.844,E2 283.2045} C_DIS
LIN {X -79.6766,Y 24.8922,Z 86,A 157.0101,B 24.9074,C -2.2222,E1 24.8474,E2 287.8112} C_DIS
LIN {X -78.0584,Y 29.5775,Z 86,A 153.5173,B 24.9067,C -2.2302,E1 24.8507,E2 291.3046} C_DIS
LIN {X -76.8517,Y 32.5853,Z 86,A 150.7392,B 24.9074,C -2.2224,E1 24.8537,E2 294.1169} C_DIS
LIN {X -75.1289,Y 36.3812,Z 86,A 147.6324,B 24.9072,C -2.2244,E1 24.8574,E2 297.2357} C_DIS
LIN {X -73.4543,Y 39.6539,Z 86,A 146.17,B 24.9042,C -2.2598,E1 24.8592,E2 298.6214} C_DIS
LIN {X -71.0944,Y 43.7437,Z 86,A 142.2495,B 24.9049,C -2.251,E1 24.8648,E2 302.5833} C_DIS
LIN {X -68.8739,Y 47.1648,Z 86,A 139.6757,B 24.9038,C -2.2647,E1 24.8688,E2 305.1372} C_DIS
LIN {X -65.3213,Y 51.9725,Z 86,A 135.5564,B 24.9029,C -2.2752,E1 24.8757,E2 309.2512} C_DIS
LIN {X -63.2924,Y 54.4258,Z 86,A 133.331,B 24.9025,C -2.2797,E1 24.8797,E2 311.476} C_DIS
LIN {X -60.3613,Y 57.6592,Z 86,A 129.9983,B 24.9026,C -2.278,E1 24.8861,E2 314.8273} C_DIS
LIN {X -57.9835,Y 60.0488,Z 86,A 128.0789,B 24.9013,C -2.2942,E1 24.8898,E2 316.7163} C_DIS
LIN {X -55.7275,Y 62.1482,Z 86,A 125.8556,B 24.9011,C -2.2961,E1 24.8944,E2 318.9439} C_DIS
LIN {X -52.1978,Y 65.1425,Z 86,A 122.508,B 24.9009,C -2.2984,E1 24.9016,E2 322.2988} C_DIS
LIN {X -49.0908,Y 67.5138,Z 86,A 119.3941,B 24.9014,C -2.2922,E1 24.9087,E2 325.4385} C_DIS
LIN {X -46.2434,Y 69.4946,Z 86,A 117.8619,B 24.899,C -2.3201,E1 24.9121,E2 326.9094} C_DIS
LIN {X -44.4717,Y 70.6421,Z 86,A 115.6349,B 24.9006,C -2.3014,E1 24.9175,E2 329.1881} C_DIS
LIN {X -41.7308,Y 72.2946,Z 86,A 114.0087,B 24.8989,C -2.321,E1 24.9213,E2 330.7724} C_DIS
LIN {X -37.3792,Y 74.6382,Z 86,A 110.3243,B 24.8991,C -2.3185,E1 24.9304,E2 334.4729} C_DIS
LIN {X -33.7793,Y 76.3355,Z 86,A 107.7864,B 24.8983,C -2.328,E1 24.9368,E2 336.9945} C_DIS
LIN {X -28.7643,Y 78.3617,Z 86,A 103.9318,B 24.8983,C -2.329,E1 24.9469,E2 340.8549} C_DIS
LIN {X -21.771,Y 80.5851,Z 86,A 99.078,B 24.8973,C -2.3399,E1 24.9598,E2 345.6913} C_DIS
LIN {X -18.4961,Y 81.3995,Z 86,A 96.6353,B 24.8973,C -2.3384,E1 24.9664,E2 348.1407} C_DIS
LIN {X -15.2433,Y 82.0715,Z 86,A 94.3518,B 24.8973,C -2.3401,E1 24.9727,E2 350.4227} C_DIS
LIN {X -11.808,Y 82.6349,Z 86,A 91.8084,B 24.8975,C -2.3373,E1 24.9797,E2 352.9749} C_DIS
LIN {X -6.9634,Y 83.1839,Z 86,A 88.992,B 24.896,C -2.3544,E1 24.9875,E2 355.7523} C_DIS
LIN {X -3.4372,Y 83.4036,Z 86,A 86.361,B 24.8964,C -2.3493,E1 24.9948,E2 358.3962} C_DIS
LIN {X 0.7912,Y 83.4709,Z 86,A 83.2013,B 24.897,C -2.3424,E1 25.0037,E2 361.5723} C_DIS
LIN {X 4.0445,Y 83.3774,Z 86,A 81.1424,B 24.8966,C -2.3477,E1 25.0094,E2 363.6181} C_DIS
LIN {X 7.0417,Y 83.1776,Z 86,A 79.0533,B 24.8966,C -2.3468,E1 25.0152,E2 365.7083} C_DIS
LIN {X 11.9832,Y 82.61,Z 86,A 75.9963,B 24.8958,C -2.3568,E1 25.0236,E2 368.7392} C_DIS
LIN {X 14.3556,Y 82.2316,Z 86,A 74.2302,B 24.8961,C -2.3528,E1 25.0285,E2 370.5133} C_DIS
LIN {X 17.9293,Y 81.5261,Z 86,A 71.4997,B 24.8968,C -2.3447,E1 25.036,E2 373.2594} C_DIS
LIN {X 21.1969,Y 80.7392,Z 86,A 69.1391,B 24.8971,C -2.3417,E1 25.0424,E2 375.6235} C_DIS
LIN {X 24.3987,Y 79.8296,Z 86,A 66.5263,B 24.8981,C -2.3302,E1 25.0495,E2 378.2592} C_DIS
LIN {X 28.6843,Y 78.3911,Z 86,A 63.4568,B 24.8983,C -2.3285,E1 25.0576,E2 381.3265} C_DIS
LIN {X 32.5295,Y 76.8752,Z 86,A 61.0979,B 24.8972,C -2.3402,E1 25.0636,E2 383.6522} C_DIS
LIN {X 35.0772,Y 75.7467,Z 86,A 58.3173,B 24.8998,C -2.3114,E1 25.0708,E2 386.4939} C_DIS
LIN {X 38.6408,Y 73.9927,Z 86,A 56.3234,B 24.8981,C -2.3304,E1 25.0756,E2 388.4375} C_DIS
LIN {X 43.3453,Y 71.3381,Z 86,A 52.0504,B 24.9001,C -2.3076,E1 25.086,E2 392.7514} C_DIS
LIN {X 46.3472,Y 69.427,Z 86,A 49.5716,B 24.9005,C -2.3026,E1 25.0918,E2 395.2339} C_DIS
LIN {X 49.274,Y 67.3797,Z 86,A 47.3856,B 24.9002,C -2.3066,E1 25.0967,E2 397.4026} C_DIS
LIN {X 52.6384,Y 64.7854,Z 86,A 44.952,B 24.8993,C -2.3165,E1 25.1019,E2 399.8038} C_DIS
LIN {X 55.0627,Y 62.7382,Z 86,A 42.8661,B 24.8994,C -2.3152,E1 25.1063,E2 401.8846} C_DIS
LIN {X 57.1511,Y 60.8416,Z 86,A 40.7842,B 24.9002,C -2.3067,E1 25.1106,E2 403.9782} C_DIS
LIN {X 60.7389,Y 57.2603,Z 86,A 37.4298,B 24.9005,C -2.3032,E1 25.1172,E2 407.3264} C_DIS
LIN {X 63.599,Y 54.0659,Z 86,A 34.4183,B 24.9012,C -2.2944,E1 25.1228,E2 410.3453} C_DIS
LIN {X 66.5473,Y 50.3935,Z 86,A 30.6522,B 24.9034,C -2.2696,E1 25.1293,E2 414.1523} C_DIS
LIN {X 68.4308,Y 47.8039,Z 86,A 28.501,B 24.9037,C -2.2656,E1 25.1328,E2 416.3025} C_DIS
LIN {X 71.7199,Y 42.7115,Z 86,A 24.8222,B 24.9033,C -2.2703,E1 25.1382,E2 419.9514} C_DIS
LIN {X 73.4255,Y 39.707,Z 86,A 21.9167,B 24.9053,C -2.2467,E1 25.1421,E2 422.8976} C_DIS
LIN {X 75.0026,Y 36.6436,Z 86,A 20.0675,B 24.9045,C -2.2568,E1 25.1444,E2 424.713} C_DIS
LIN {X 76.4708,Y 33.469,Z 86,A 17.3882,B 24.9058,C -2.241,E1 25.1474,E2 427.4152} C_DIS
LIN {X 78.0384,Y 29.6303,Z 86,A 15.0224,B 24.9052,C -2.2484,E1 25.1498,E2 429.7502} C_DIS
LIN {X 79.1957,Y 26.3832,Z 86,A 12.7178,B 24.9056,C -2.2435,E1 25.152,E2 432.0536} C_DIS
LIN {X 80.1059,Y 23.4749,Z 86,A 10.4984,B 24.9065,C -2.233,E1 25.1538,E2 434.285} C_DIS
LIN {X 80.9922,Y 20.2089,Z 86,A 8.2588,B 24.9068,C -2.2287,E1 25.1553,E2 436.5219} C_DIS
LIN {X 81.6396,Y 17.4088,Z 86,A 5.9163,B 24.9083,C -2.2104,E1 25.1568,E2 438.8939} C_DIS
LIN {X 82.2039,Y 14.5096,Z 86,A 3.4055,B 24.9102,C -2.1883,E1 25.158,E2 441.4422} C_DIS
LIN {X 82.8232,Y 10.4098,Z 86,A 1.6724,B 24.9079,C -2.216,E1 25.1586,E2 443.0997} C_DIS
LIN {X 83.0796,Y 8.1192,Z 86,A -0.8924,B 24.911,C -2.1786,E1 25.1593,E2 445.7377} C_DIS
LIN {X 83.3619,Y 4.3366,Z 86,A -3.256,B 24.911,C -2.1782,E1 25.1597,E2 448.0882} C_DIS
LIN {X 83.4701,Y -0.9211,Z 86,A -6.385,B 24.9107,C -2.1825,E1 25.1597,E2 451.1884} C_DIS
LIN {X 83.2681,Y -5.8671,Z 86,A -9.9214,B 24.9119,C -2.167,E1 25.1592,E2 454.7403} C_DIS
LIN {X 82.9028,Y -9.7505,Z 86,A -12.3529,B 24.9119,C -2.1666,E1 25.1585,E2 457.1584} C_DIS
LIN {X 82.4667,Y -12.9312,Z 86,A -14.4943,B 24.9124,C -2.1617,E1 25.1577,E2 459.2989} C_DIS
LIN {X 81.6105,Y -17.5422,Z 86,A -18.1196,B 24.9143,C -2.138,E1 25.1557,E2 462.9588} C_DIS
LIN {X 79.9474,Y -24.0092,Z 86,A -22.424,B 24.9147,C -2.1328,E1 25.1525,E2 467.2507} C_DIS
LIN {X 78.0862,Y -29.5042,Z 86,A -26.1997,B 24.9151,C -2.1274,E1 25.1491,E2 471.018} C_DIS
LIN {X 77.1199,Y -31.9485,Z 86,A -28.691,B 24.9174,C -2.0992,E1 25.1464,E2 473.5621} C_DIS
LIN {X 75.721,Y -35.1325,Z 86,A -30.4878,B 24.9164,C -2.1115,E1 25.1443,E2 475.3202} C_DIS
LIN {X 74.4102,Y -37.8299,Z 86,A -32.4833,B 24.9167,C -2.1075,E1 25.1418,E2 477.3145} C_DIS
LIN {X 72.4763,Y -41.4146,Z 86,A -35.0879,B 24.9169,C -2.1056,E1 25.1384,E2 479.9099} C_DIS
LIN {X 71.2437,Y -43.5007,Z 86,A -36.9067,B 24.9176,C -2.0957,E1 25.1357,E2 481.7427} C_DIS
LIN {X 69.6097,Y -46.0701,Z 86,A -38.9474,B 24.918,C -2.0915,E1 25.1326,E2 483.7832} C_DIS
LIN {X 67.317,Y -49.3591,Z 86,A -41.6966,B 24.9185,C -2.0841,E1 25.1282,E2 486.5365} C_DIS
LIN {X 64.8741,Y -52.529,Z 86,A -44.8479,B 24.9201,C -2.0636,E1 25.1227,E2 489.7214} C_DIS
LIN {X 62.5677,Y -55.2579,Z 86,A -48.0494,B 24.9225,C -2.0332,E1 25.1166,E2 492.9803} C_DIS
LIN {X 59.0056,Y -59.0468,Z 86,A -51.5069,B 24.9229,C -2.0282,E1 25.1098,E2 496.4352} C_DIS
LIN {X 55.4583,Y -62.3892,Z 86,A -53.5152,B 24.9202,C -2.0634,E1 25.1059,E2 498.352} C_DIS
LIN {X 51.3251,Y -65.8322,Z 86,A -57.3769,B 24.9212,C -2.0497,E1 25.0975,E2 502.2314} C_DIS
LIN {X 48.7978,Y -67.7265,Z 86,A -59.5514,B 24.9216,C -2.045,E1 25.0926,E2 504.4093} C_DIS
LIN {X 46.5678,Y -69.2782,Z 86,A -61.4945,B 24.9221,C -2.0388,E1 25.0881,E2 506.3605} C_DIS
LIN {X 42.1999,Y -72.0223,Z 86,A -65.1551,B 24.9229,C -2.0284,E1 25.0793,E2 510.0342} C_DIS
LIN {X 38.945,Y -73.8325,Z 86,A -68.0651,B 24.924,C -2.0128,E1 25.0721,E2 512.9728} C_DIS
LIN {X 36.0573,Y -75.285,Z 86,A -69.7344,B 24.923,C -2.0266,E1 25.068,E2 514.6051} C_DIS
LIN {X 32.0739,Y -77.0672,Z 86,A -72.8312,B 24.9236,C -2.0189,E1 25.0601,E2 517.7125} C_DIS
LIN {X 29.8669,Y -77.9488,Z 86,A -74.3582,B 24.9235,C -2.02,E1 25.0561,E2 519.2336} C_DIS
LIN {X 25.3452,Y -79.5343,Z 86,A -77.8287,B 24.9242,C -2.0102,E1 25.0469,E2 522.7205} C_DIS
LIN {X 21.32,Y -80.707,Z 86,A -80.5866,B 24.9242,C -2.0108,E1 25.0395,E2 525.4725} C_DIS
LIN {X 16.9734,Y -81.7306,Z 86,A -84.1308,B 24.9255,C -1.9933,E1 25.0297,E2 529.0535} C_DIS
LIN {X 13.7124,Y -82.3403,Z 86,A -85.7308,B 24.9241,C -2.0123,E1 25.0254,E2 530.6067} C_DIS
LIN {X 10.9262,Y -82.7563,Z 86,A -87.8081,B 24.9245,C -2.0066,E1 25.0197,E2 532.6958} C_DIS
LIN {X 6.2191,Y -83.2432,Z 86,A -91.1619,B 24.9249,C -2.0017,E1 25.0103,E2 536.0593} C_DIS
LIN {X 2.5188,Y -83.4362,Z 86,A -93.5121,B 24.9245,C -2.0066,E1 25.0038,E2 538.3971} C_DIS
LIN {X 0.5322,Y -83.4702,Z 86,A -94.7144,B 24.9242,C -2.0112,E1 25.0005,E2 539.5883} C_DIS
Enddeposition()
LIN {X 0.5322,Y -83.4702,Z 86,A -94.7144,B 24.9242,C -2.0112,E1 25.0005,E2 539.5883} C_DIS
Startdeposition()
$VEL.CP = VEL_PRINT
LIN {X 1.0779,Y -82.5613,Z 86,A -93.5127,B 24.921,C -2.052,E1 25.0041,E2 538.29} C_DIS
LIN {X 4.2222,Y -82.4598,Z 86,A -91.0488,B 24.9203,C -2.0615,E1 25.011,E2 535.8044} C_DIS
LIN {X 8.5809,Y -82.12,Z 86,A -88.4577,B 24.9212,C -2.0494,E1 25.0181,E2 533.2434} C_DIS
LIN {X 11.2055,Y -81.8043,Z 86,A -86.3783,B 24.9206,C -2.0581,E1 25.0239,E2 531.1449} C_DIS
LIN {X 14.6216,Y -81.2622,Z 86,A -83.8605,B 24.9201,C -2.0636,E1 25.0309,E2 528.6167} C_DIS
LIN {X 19.0676,Y -80.3368,Z 86,A -80.8223,B 24.9201,C -2.063,E1 25.0392,E2 525.5842} C_DIS
LIN {X 23.495,Y -79.1538,Z 86,A -77.913,B 24.9206,C -2.0579,E1 25.047,E2 522.6917} C_DIS
LIN {X 27.3104,Y -77.9197,Z 86,A -74.6035,B 24.919,C -2.078,E1 25.0558,E2 519.341} C_DIS
LIN {X 32.4991,Y -75.9022,Z 86,A -71.0616,B 24.9194,C -2.0732,E1 25.0649,E2 515.8185} C_DIS
LIN {X 35.4864,Y -74.5528,Z 86,A -68.9594,B 24.9195,C -2.0713,E1 25.0702,E2 513.7263} C_DIS
LIN {X 38.5403,Y -73.0204,Z 86,A -66.8535,B 24.9199,C -2.0668,E1 25.0754,E2 511.6369} C_DIS
LIN {X 40.4469,Y -71.9821,Z 86,A -65.1077,B 24.9191,C -2.077,E1 25.0797,E2 509.8719} C_DIS
LIN {X 43.6661,Y -70.0757,Z 86,A -62.9079,B 24.9197,C -2.0691,E1 25.0849,E2 507.6976} C_DIS
LIN {X 45.5007,Y -68.8986,Z 86,A -60.915,B 24.9183,C -2.0875,E1 25.0897,E2 505.6679} C_DIS
LIN {X 48.2977,Y -66.9689,Z 86,A -58.6678,B 24.9182,C -2.0886,E1 25.0948,E2 503.4256} C_DIS
LIN {X 51.2965,Y -64.6994,Z 86,A -55.5279,B 24.9164,C -2.1115,E1 25.1018,E2 500.2432} C_DIS
LIN {X 54.934,Y -61.6411,Z 86,A -52.7409,B 24.9171,C -2.1022,E1 25.1076,E2 497.4891} C_DIS
LIN {X 57.7388,Y -59.023,Z 86,A -49.9728,B 24.9163,C -2.112,E1 25.1133,E2 494.7093} C_DIS
LIN {X 61.3807,Y -55.2248,Z 86,A -46.8213,B 24.9169,C -2.1047,E1 25.1193,E2 491.5888} C_DIS
LIN {X 63.7873,Y -52.4282,Z 86,A -43.204,B 24.9136,C -2.1461,E1 25.1259,E2 487.8902} C_DIS
LIN {X 66.0629,Y -49.5281,Z 86,A -41.0998,B 24.9143,C -2.1379,E1 25.1294,E2 485.8153} C_DIS
LIN {X 68.1658,Y -46.5928,Z 86,A -38.8074,B 24.9143,C -2.1377,E1 25.133,E2 483.5347} C_DIS
LIN {X 70.0627,Y -43.6871,Z 86,A -36.4132,B 24.9138,C -2.1441,E1 25.1366,E2 481.1376} C_DIS
LIN {X 71.9067,Y -40.5819,Z 86,A -33.9769,B 24.9134,C -2.149,E1 25.14,E2 478.7023} C_DIS
LIN {X 72.9706,Y -38.635,Z 86,A -32.5003,B 24.9132,C -2.1514,E1 25.142,E2 477.2278} C_DIS
LIN {X 74.2927,Y -36.0279,Z 86,A -30.5366,B 24.9129,C -2.1552,E1 25.1444,E2 475.2655} C_DIS
LIN {X 76.497,Y -31.0731,Z 86,A -26.8142,B 24.9121,C -2.1652,E1 25.1486,E2 471.5399} C_DIS
LIN {X 77.845,Y -27.5232,Z 86,A -23.8062,B 24.9104,C -2.1857,E1 25.1515,E2 468.5002} C_DIS
LIN {X 78.9343,Y -24.2231,Z 86,A -20.7062,B 24.9078,C -2.2164,E1 25.1541,E2 465.3454} C_DIS
LIN {X 80.1656,Y -19.77,Z 86,A -18.3773,B 24.9095,C -2.197,E1 25.1556,E2 463.0759} C_DIS
LIN {X 81.0565,Y -15.722,Z 86,A -15.6838,B 24.9092,C -2.2,E1 25.1571,E2 460.3909} C_DIS
LIN {X 81.6622,Y -12.1981,Z 86,A -13.0338,B 24.9081,C -2.2135,E1 25.1583,E2 457.7246} C_DIS
LIN {X 82.096,Y -8.8107,Z 86,A -10.8819,B 24.9081,C -2.2138,E1 25.159,E2 455.5847} C_DIS
LIN {X 82.3582,Y -5.8786,Z 86,A -8.6139,B 24.9069,C -2.2279,E1 25.1595,E2 453.2969} C_DIS
LIN {X 82.5235,Y -2.6883,Z 86,A -6.5919,B 24.9069,C -2.2285,E1 25.1597,E2 451.2856} C_DIS
LIN {X 82.5637,Y 0.7586,Z 86,A -4.1967,B 24.9062,C -2.2362,E1 25.1597,E2 448.8864} C_DIS
LIN {X 82.4422,Y 4.5407,Z 86,A -1.3778,B 24.9049,C -2.251,E1 25.1594,E2 446.0492} C_DIS
LIN {X 82.1351,Y 8.4369,Z 86,A 1.0503,B 24.905,C -2.2501,E1 25.1588,E2 443.6377} C_DIS
LIN {X 81.7642,Y 11.4878,Z 86,A 3.58,B 24.9033,C -2.27,E1 25.1578,E2 441.0759} C_DIS
LIN {X 81.2158,Y 14.8792,Z 86,A 5.5631,B 24.9038,C -2.2641,E1 25.1569,E2 439.1184} C_DIS
LIN {X 80.7802,Y 17.0919,Z 86,A 7.1392,B 24.9034,C -2.2692,E1 25.156,E2 437.5393} C_DIS
LIN {X 80.1101,Y 19.9976,Z 86,A 9.1834,B 24.9029,C -2.2747,E1 25.1547,E2 435.4939} C_DIS
LIN {X 79.3785,Y 22.7254,Z 86,A 11.037,B 24.9027,C -2.2771,E1 25.1533,E2 433.6453} C_DIS
LIN {X 78.5088,Y 25.568,Z 86,A 13.8076,B 24.9002,C -2.3068,E1 25.1509,E2 430.8204} C_DIS
Enddeposition()
END
